LIN {X 0,Y 305.806,Z 453.018,A -85,B 0,C 180,E1 -16012.074,E2 -16012.074} C_VEL
LIN {X 0,Y 305.684,Z 453.026,A -85,B 0,C 180,E1 -16014.724,E2 -16014.724} C_VEL
LIN {X 0,Y 305.951,Z 452.995,A -85,B 0,C 180,E1 -16018.684,E2 -16018.684} C_VEL
LIN {X 0,Y 305.951,Z 452.99,A -85,B 0,C 180,E1 -16021.317,E2 -16021.317} C_VEL
LIN {X 0,Y 305.684,Z 453.027,A -85,B 0,C 180,E1 -16025.277,E2 -16025.277} C_VEL
LIN {X 0,Y 305.806,Z 453.011,A -85,B 0,C 180,E1 -16027.926,E2 -16027.926} C_VEL
LIN {X 0,Y 305.597,Z 453.04,A -85,B 0,C 180,E1 -16031.946,E2 -16031.946} C_VEL
LIN {X 0,Y 305.632,Z 453.04,A -85,B 0,C 180,E1 -16035.036,E2 -16035.036} C_VEL
LIN {X 0,Y 305.572,Z 453.044,A -85,B 0,C 180,E1 -16039.446,E2 -16039.446} C_VEL
LIN {X 0,Y 305.485,Z 453.061,A -85,B 0,C 180,E1 -16043.042,E2 -16043.042} C_VEL
LIN {X 0,Y 305.527,Z 453.043,A -85,B 0,C 180,E1 -16046.74,E2 -16046.74} C_VEL
LIN {X 0,Y 305.538,Z 453.238,A -85,B 0,C 180,E1 -16047.227,E2 -16047.227} C_VEL
LIN {X 0,Y 305.899,Z 454.626,A -85,B 0,C 180,E1 -16047.726,E2 -16047.726} C_VEL
LIN {X 0,Y 308.583,Z 458.796,A -85,B 0,C 180,E1 -16048.341,E2 -16048.341} C_VEL
LIN {X 0,Y 315.737,Z 470.32,A -85,B 0,C 180,E1 -16049.906,E2 -16049.906} C_VEL
LIN {X 0,Y 324.283,Z 485.614,A -85,B 0,C 180,E1 -16051.666,E2 -16051.666} C_VEL
LIN {X 0,Y 332.768,Z 503.328,A -85,B 0,C 180,E1 -16053.337,E2 -16053.337} C_VEL
LIN {X 0,Y 333.643,Z 505.601,A -85,B 0,C 180,E1 -16053.514,E2 -16053.514} C_VEL
LIN {X 0,Y 329.127,Z 618.858,A -85,B 0,C 180,E1 -16056.067,E2 -16056.067} C_VEL
LIN {X 0,Y 327.823,Z 634.58,A -85,B 0,C 180,E1 -16056.652,E2 -16056.652} C_VEL
LIN {X 0,Y 326.147,Z 650.125,A -85,B 0,C 180,E1 -16057.511,E2 -16057.511} C_VEL
LIN {X 0,Y 324.166,Z 664.525,A -85,B 0,C 180,E1 -16058.572,E2 -16058.572} C_VEL
LIN {X 0,Y 321.994,Z 677.479,A -85,B 0,C 180,E1 -16059.769,E2 -16059.769} C_VEL
LIN {X 0,Y 319.469,Z 690.779,A -85,B 0,C 180,E1 -16061.298,E2 -16061.298} C_VEL
LIN {X 0,Y 316.932,Z 702.653,A -85,B 0,C 180,E1 -16062.966,E2 -16062.966} C_VEL
LIN {X 0,Y 314.485,Z 713.443,A -85,B 0,C 180,E1 -16064.804,E2 -16064.804} C_VEL
LIN {X 0,Y 311.875,Z 724.247,A -85,B 0,C 180,E1 -16067.027,E2 -16067.027} C_VEL
LIN {X 0,Y 309.653,Z 733.163,A -85,B 0,C 180,E1 -16069.27,E2 -16069.27} C_VEL
LIN {X 0,Y 307.598,Z 741.721,A -85,B 0,C 180,E1 -16071.912,E2 -16071.912} C_VEL
LIN {X 0,Y 306.244,Z 747.624,A -85,B 0,C 180,E1 -16074.184,E2 -16074.184} C_VEL
LIN {X 0,Y 305.187,Z 752.434,A -85,B 0,C 180,E1 -16076.45,E2 -16076.45} C_VEL
LIN {X 0,Y 304.545,Z 756.122,A -85,B 0,C 180,E1 -16078.634,E2 -16078.634} C_VEL
LIN {X 0,Y 303.801,Z 759.699,A -85,B 0,C 180,E1 -16081.532,E2 -16081.532} C_VEL
LIN {X 0,Y 303.421,Z 761.961,A -85,B 0,C 180,E1 -16084.602,E2 -16084.602} C_VEL
LIN {X 0,Y 303.279,Z 762.664,A -85,B 0,C 180,E1 -16087.963,E2 -16087.963} C_VEL
LIN {X 0,Y 303.416,Z 761.698,A -85,B 0,C 180,E1 -16091.079,E2 -16091.079} C_VEL
LIN {X 0,Y 303.711,Z 759.497,A -85,B 0,C 180,E1 -16093.879,E2 -16093.879} C_VEL
LIN {X 0,Y 304.241,Z 756.014,A -85,B 0,C 180,E1 -16096.645,E2 -16096.645} C_VEL
LIN {X 0,Y 304.998,Z 751.21,A -85,B 0,C 180,E1 -16099.378,E2 -16099.378} C_VEL
LIN {X 0,Y 306.144,Z 744.971,A -85,B 0,C 180,E1 -16102.084,E2 -16102.084} C_VEL
LIN {X 0,Y 307.774,Z 737.108,A -85,B 0,C 180,E1 -16104.76,E2 -16104.76} C_VEL
LIN {X 0,Y 309.611,Z 728.336,A -85,B 0,C 180,E1 -16107.173,E2 -16107.173} C_VEL
LIN {X 0,Y 311.717,Z 718.677,A -85,B 0,C 180,E1 -16109.355,E2 -16109.355} C_VEL
LIN {X 0,Y 313.828,Z 708.408,A -85,B 0,C 180,E1 -16111.284,E2 -16111.284} C_VEL
LIN {X 0,Y 316.165,Z 696.881,A -85,B 0,C 180,E1 -16113.075,E2 -16113.075} C_VEL
LIN {X 0,Y 318.618,Z 683.799,A -85,B 0,C 180,E1 -16114.745,E2 -16114.745} C_VEL
LIN {X 0,Y 320.826,Z 670.4,A -85,B 0,C 180,E1 -16116.131,E2 -16116.131} C_VEL
LIN {X 0,Y 322.851,Z 655.629,A -85,B 0,C 180,E1 -16117.348,E2 -16117.348} C_VEL
LIN {X 0,Y 324.432,Z 641.335,A -85,B 0,C 180,E1 -16118.252,E2 -16118.252} C_VEL
LIN {X 0,Y 325.776,Z 625.914,A -85,B 0,C 180,E1 -16118.96,E2 -16118.96} C_VEL
LIN {X 0,Y 326.618,Z 609.669,A -85,B 0,C 180,E1 -16119.444,E2 -16119.444} C_VEL
LIN {X 0,Y 330.36,Z 503.226,A -85,B 0,C 180,E1 -16121.792,E2 -16121.792} C_VEL
LIN {X 0,Y 322.753,Z 486.044,A -85,B 0,C 180,E1 -16123.098,E2 -16123.098} C_VEL
LIN {X 0,Y 312.977,Z 466.729,A -85,B 0,C 180,E1 -16124.819,E2 -16124.819} C_VEL
LIN {X 0,Y 308.703,Z 459.164,A -85,B 0,C 180,E1 -16125.584,E2 -16125.584} C_VEL
LIN {X 0,Y 307.211,Z 456.721,A -85,B 0,C 180,E1 -16125.853,E2 -16125.853} C_VEL
LIN {X 0,Y 305.8,Z 454.164,A -85,B 0,C 180,E1 -16126.117,E2 -16126.117} C_VEL
LIN {X 0,Y 305.59,Z 453.042,A -85,B 0,C 180,E1 -16126.235,E2 -16126.235} C_VEL
LIN {X 0,Y 305.585,Z 453.048,A -85,B 0,C 180,E1 -16129.448,E2 -16129.448} C_VEL
LIN {X 0,Y 305.495,Z 453.058,A -85,B 0,C 180,E1 -16133.042,E2 -16133.042} C_VEL
LIN {X 0,Y 305.518,Z 453.047,A -85,B 0,C 180,E1 -16135.169,E2 -16135.169} C_VEL
LIN {X 0,Y 304.872,Z 453.135,A -85,B 0,C 180,E1 -16136.269,E2 -16136.269} C_VEL
LIN {X 0,Y 301.967,Z 453.492,A -85,B 0,C 180,E1 -16138.058,E2 -16138.058} C_VEL
LIN {X 0,Y 299.498,Z 453.8,A -85,B 0,C 180,E1 -16139.51,E2 -16139.51} C_VEL
LIN {X 0,Y 298.461,Z 453.933,A -85,B 0,C 180,E1 -16140.636,E2 -16140.636} C_VEL
LIN {X 0,Y 298.391,Z 453.937,A -85,B 0,C 180,E1 -16141.017,E2 -16141.017} C_VEL
LIN {X 0,Y 298.431,Z 453.936,A -85,B 0,C 180,E1 -16144.487,E2 -16144.487} C_VEL
LIN {X 0,Y 298.418,Z 453.921,A -85,B 0,C 180,E1 -16147.758,E2 -16147.758} C_VEL
LIN {X 0,Y 298.416,Z 453.939,A -85,B 0,C 180,E1 -16151.257,E2 -16151.257} C_VEL
LIN {X 0,Y 298.357,Z 453.943,A -85,B 0,C 180,E1 -16155.035,E2 -16155.035} C_VEL
LIN {X 0,Y 298.435,Z 453.934,A -85,B 0,C 180,E1 -16156.926,E2 -16156.926} C_VEL
LIN {X 0,Y 298.428,Z 453.936,A -85,B 0,C 180,E1 -16161.001,E2 -16161.001} C_VEL
LIN {X 0,Y 298.434,Z 453.921,A -85,B 0,C 180,E1 -16163.932,E2 -16163.932} C_VEL
LIN {X 0,Y 298.396,Z 453.937,A -85,B 0,C 180,E1 -16167.983,E2 -16167.983} C_VEL
LIN {X 0,Y 298.461,Z 453.926,A -85,B 0,C 180,E1 -16171.904,E2 -16171.904} C_VEL
LIN {X 0,Y 298.486,Z 453.925,A -85,B 0,C 180,E1 -16174.924,E2 -16174.924} C_VEL
LIN {X 0,Y 298.443,Z 453.932,A -85,B 0,C 180,E1 -16179.314,E2 -16179.314} C_VEL
LIN {X 0,Y 298.539,Z 453.91,A -85,B 0,C 180,E1 -16182.179,E2 -16182.179} C_VEL
LIN {X 0,Y 298.595,Z 453.905,A -85,B 0,C 180,E1 -16184.994,E2 -16184.994} C_VEL
LIN {X 0,Y 298.595,Z 453.902,A -85,B 0,C 180,E1 -16189.146,E2 -16189.146} C_VEL
LIN {X 0,Y 298.759,Z 453.885,A -85,B 0,C 180,E1 -16191.886,E2 -16191.886} C_VEL
LIN {X 0,Y 298.661,Z 453.904,A -85,B 0,C 180,E1 -16194.599,E2 -16194.599} C_VEL
LIN {X 0,Y 298.924,Z 453.867,A -85,B 0,C 180,E1 -16198.652,E2 -16198.652} C_VEL
LIN {X 0,Y 298.924,Z 453.875,A -85,B 0,C 180,E1 -16201.347,E2 -16201.347} C_VEL
LIN {X 0,Y 298.798,Z 453.883,A -85,B 0,C 180,E1 -16206.754,E2 -16206.754} C_VEL
LIN {X 0,Y 298.681,Z 453.902,A -85,B 0,C 180,E1 -16209.48,E2 -16209.48} C_VEL
LIN {X 0,Y 298.552,Z 453.909,A -85,B 0,C 180,E1 -16213.615,E2 -16213.615} C_VEL
LIN {X 0,Y 298.549,Z 453.918,A -85,B 0,C 180,E1 -16216.408,E2 -16216.408} C_VEL
LIN {X 0,Y 298.512,Z 453.911,A -85,B 0,C 180,E1 -16219.654,E2 -16219.654} C_VEL
LIN {X 0,Y 298.458,Z 453.931,A -85,B 0,C 180,E1 -16223.597,E2 -16223.597} C_VEL
LIN {X 0,Y 298.49,Z 453.928,A -85,B 0,C 180,E1 -16226.574,E2 -16226.574} C_VEL
LIN {X 0,Y 298.421,Z 453.938,A -85,B 0,C 180,E1 -16229.641,E2 -16229.641} C_VEL
LIN {X 0,Y 298.396,Z 453.939,A -85,B 0,C 180,E1 -16232.8,E2 -16232.8} C_VEL
LIN {X 0,Y 298.465,Z 453.931,A -85,B 0,C 180,E1 -16236.812,E2 -16236.812} C_VEL
LIN {X 0,Y 298.413,Z 453.938,A -85,B 0,C 180,E1 -16241.093,E2 -16241.093} C_VEL
LIN {X 0,Y 298.417,Z 453.939,A -85,B 0,C 180,E1 -16245.047,E2 -16245.047} C_VEL
LIN {X 0,Y 298.479,Z 454.134,A -85,B 0,C 180,E1 -16247.17,E2 -16247.17} C_VEL
LIN {X 0,Y 301.356,Z 464.027,A -85,B 0,C 180,E1 -16250.318,E2 -16250.318} C_VEL
LIN {X 0,Y 302.376,Z 467.643,A -85,B 0,C 180,E1 -16251.412,E2 -16251.412} C_VEL
LIN {X 0,Y 311.581,Z 486.103,A -85,B 0,C 180,E1 -16253.155,E2 -16253.155} C_VEL
LIN {X 0,Y 320.741,Z 506.44,A -85,B 0,C 180,E1 -16254.821,E2 -16254.821} C_VEL
LIN {X 0,Y 321.941,Z 509.914,A -85,B 0,C 180,E1 -16255.052,E2 -16255.052} C_VEL
LIN {X 0,Y 323.888,Z 521.419,A -85,B 0,C 180,E1 -16255.577,E2 -16255.577} C_VEL
LIN {X 0,Y 319.755,Z 634.882,A -85,B 0,C 180,E1 -16258.163,E2 -16258.163} C_VEL
LIN {X 0,Y 318.413,Z 650.708,A -85,B 0,C 180,E1 -16258.755,E2 -16258.755} C_VEL
LIN {X 0,Y 316.681,Z 665.871,A -85,B 0,C 180,E1 -16259.584,E2 -16259.584} C_VEL
LIN {X 0,Y 314.806,Z 679.599,A -85,B 0,C 180,E1 -16260.584,E2 -16260.584} C_VEL
LIN {X 0,Y 312.607,Z 693.075,A -85,B 0,C 180,E1 -16261.828,E2 -16261.828} C_VEL
LIN {X 0,Y 310.241,Z 705.501,A -85,B 0,C 180,E1 -16263.241,E2 -16263.241} C_VEL
LIN {X 0,Y 307.679,Z 718.163,A -85,B 0,C 180,E1 -16265.002,E2 -16265.002} C_VEL
LIN {X 0,Y 305.207,Z 729.668,A -85,B 0,C 180,E1 -16266.954,E2 -16266.954} C_VEL
LIN {X 0,Y 303.224,Z 739.352,A -85,B 0,C 180,E1 -16268.945,E2 -16268.945} C_VEL
LIN {X 0,Y 301.062,Z 748.848,A -85,B 0,C 180,E1 -16271.277,E2 -16271.277} C_VEL
LIN {X 0,Y 299.473,Z 756.751,A -85,B 0,C 180,E1 -16273.643,E2 -16273.643} C_VEL
LIN {X 0,Y 298.063,Z 764.116,A -85,B 0,C 180,E1 -16276.361,E2 -16276.361} C_VEL
LIN {X 0,Y 297.147,Z 769.933,A -85,B 0,C 180,E1 -16279.093,E2 -16279.093} C_VEL
LIN {X 0,Y 296.711,Z 774.37,A -85,B 0,C 180,E1 -16281.829,E2 -16281.829} C_VEL
LIN {X 0,Y 296.511,Z 777.526,A -85,B 0,C 180,E1 -16284.559,E2 -16284.559} C_VEL
LIN {X 0,Y 296.515,Z 779.449,A -85,B 0,C 180,E1 -16287.282,E2 -16287.282} C_VEL
LIN {X 0,Y 296.518,Z 780.155,A -85,B 0,C 180,E1 -16289.999,E2 -16289.999} C_VEL
LIN {X 0,Y 296.517,Z 779.71,A -85,B 0,C 180,E1 -16292.716,E2 -16292.716} C_VEL
LIN {X 0,Y 296.51,Z 778.111,A -85,B 0,C 180,E1 -16295.44,E2 -16295.44} C_VEL
LIN {X 0,Y 296.706,Z 775.339,A -85,B 0,C 180,E1 -16298.17,E2 -16298.17} C_VEL
LIN {X 0,Y 297.183,Z 771.322,A -85,B 0,C 180,E1 -16300.905,E2 -16300.905} C_VEL
LIN {X 0,Y 298.133,Z 765.949,A -85,B 0,C 180,E1 -16303.634,E2 -16303.634} C_VEL
LIN {X 0,Y 299.517,Z 759.127,A -85,B 0,C 180,E1 -16306.353,E2 -16306.353} C_VEL
LIN {X 0,Y 301.511,Z 750.68,A -85,B 0,C 180,E1 -16309.045,E2 -16309.045} C_VEL
LIN {X 0,Y 303.455,Z 743.047,A -85,B 0,C 180,E1 -16311.036,E2 -16311.036} C_VEL
LIN {X 0,Y 305.947,Z 732.701,A -85,B 0,C 180,E1 -16313.307,E2 -16313.307} C_VEL
LIN {X 0,Y 308.532,Z 721.78,A -85,B 0,C 180,E1 -16315.283,E2 -16315.283} C_VEL
LIN {X 0,Y 311.268,Z 710.08,A -85,B 0,C 180,E1 -16317.025,E2 -16317.025} C_VEL
LIN {X 0,Y 314,Z 697.34,A -85,B 0,C 180,E1 -16318.581,E2 -16318.581} C_VEL
LIN {X 0,Y 316.67,Z 683.092,A -85,B 0,C 180,E1 -16319.984,E2 -16319.984} C_VEL
LIN {X 0,Y 318.926,Z 668.805,A -85,B 0,C 180,E1 -16321.095,E2 -16321.095} C_VEL
LIN {X 0,Y 320.944,Z 653.611,A -85,B 0,C 180,E1 -16321.981,E2 -16321.981} C_VEL
LIN {X 0,Y 322.504,Z 638.634,A -85,B 0,C 180,E1 -16322.592,E2 -16322.592} C_VEL
LIN {X 0,Y 323.448,Z 620.384,A -85,B 0,C 180,E1 -16323.087,E2 -16323.087} C_VEL
LIN {X 0,Y 326.87,Z 535.782,A -85,B 0,C 180,E1 -16324.996,E2 -16324.996} C_VEL
LIN {X 0,Y 327.351,Z 521.586,A -85,B 0,C 180,E1 -16325.33,E2 -16325.33} C_VEL
LIN {X 0,Y 325.679,Z 511.869,A -85,B 0,C 180,E1 -16325.833,E2 -16325.833} C_VEL
LIN {X 0,Y 319.096,Z 497.086,A -85,B 0,C 180,E1 -16327.216,E2 -16327.216} C_VEL
LIN {X 0,Y 312.441,Z 483.929,A -85,B 0,C 180,E1 -16328.658,E2 -16328.658} C_VEL
LIN {X 0,Y 306.561,Z 473.529,A -85,B 0,C 180,E1 -16329.986,E2 -16329.986} C_VEL
LIN {X 0,Y 302.358,Z 466.202,A -85,B 0,C 180,E1 -16331.005,E2 -16331.005} C_VEL
LIN {X 0,Y 299.851,Z 458.407,A -85,B 0,C 180,E1 -16333.886,E2 -16333.886} C_VEL
LIN {X 0,Y 298.414,Z 453.93,A -85,B 0,C 180,E1 -16335.699,E2 -16335.699} C_VEL
LIN {X 0,Y 298.407,Z 453.942,A -85,B 0,C 180,E1 -16338.906,E2 -16338.906} C_VEL
LIN {X 0,Y 298.44,Z 453.936,A -85,B 0,C 180,E1 -16343.192,E2 -16343.192} C_VEL
LIN {X 0,Y 298.389,Z 453.936,A -85,B 0,C 180,E1 -16347.199,E2 -16347.199} C_VEL
LIN {X 0,Y 298.421,Z 453.934,A -85,B 0,C 180,E1 -16350.616,E2 -16350.616} C_VEL
LIN {X 0,Y 298.472,Z 453.925,A -85,B 0,C 180,E1 -16353.476,E2 -16353.476} C_VEL
LIN {X 0,Y 298.428,Z 453.931,A -85,B 0,C 180,E1 -16356.697,E2 -16356.697} C_VEL
LIN {X 0,Y 298.533,Z 453.922,A -85,B 0,C 180,E1 -16360.757,E2 -16360.757} C_VEL
LIN {X 0,Y 298.587,Z 453.917,A -85,B 0,C 180,E1 -16364.995,E2 -16364.995} C_VEL
LIN {X 0,Y 298.589,Z 453.915,A -85,B 0,C 180,E1 -16369.147,E2 -16369.147} C_VEL
LIN {X 0,Y 298.752,Z 453.895,A -85,B 0,C 180,E1 -16371.886,E2 -16371.886} C_VEL
LIN {X 0,Y 298.655,Z 453.901,A -85,B 0,C 180,E1 -16374.599,E2 -16374.599} C_VEL
LIN {X 0,Y 298.917,Z 453.871,A -85,B 0,C 180,E1 -16378.653,E2 -16378.653} C_VEL
LIN {X 0,Y 298.917,Z 453.866,A -85,B 0,C 180,E1 -16381.348,E2 -16381.348} C_VEL
LIN {X 0,Y 298.791,Z 453.891,A -85,B 0,C 180,E1 -16386.754,E2 -16386.754} C_VEL
LIN {X 0,Y 298.674,Z 453.906,A -85,B 0,C 180,E1 -16389.481,E2 -16389.481} C_VEL
LIN {X 0,Y 298.546,Z 453.918,A -85,B 0,C 180,E1 -16393.616,E2 -16393.616} C_VEL
LIN {X 0,Y 298.543,Z 453.919,A -85,B 0,C 180,E1 -16396.409,E2 -16396.409} C_VEL
LIN {X 0,Y 298.507,Z 453.925,A -85,B 0,C 180,E1 -16399.656,E2 -16399.656} C_VEL
LIN {X 0,Y 298.452,Z 453.935,A -85,B 0,C 180,E1 -16403.599,E2 -16403.599} C_VEL
LIN {X 0,Y 298.529,Z 454.023,A -85,B 0,C 180,E1 -16406.054,E2 -16406.054} C_VEL
LIN {X 0,Y 298.682,Z 454.861,A -85,B 0,C 180,E1 -16406.373,E2 -16406.373} C_VEL
LIN {X 0,Y 299.971,Z 457.462,A -85,B 0,C 180,E1 -16406.716,E2 -16406.716} C_VEL
LIN {X 0,Y 302.219,Z 460.449,A -85,B 0,C 180,E1 -16407.247,E2 -16407.247} C_VEL
LIN {X 0,Y 306.435,Z 466.935,A -85,B 0,C 180,E1 -16408.232,E2 -16408.232} C_VEL
LIN {X 0,Y 312.861,Z 477.582,A -85,B 0,C 180,E1 -16409.668,E2 -16409.668} C_VEL
LIN {X 0,Y 320.325,Z 491.438,A -85,B 0,C 180,E1 -16411.256,E2 -16411.256} C_VEL
LIN {X 0,Y 327.895,Z 507.518,A -85,B 0,C 180,E1 -16412.803,E2 -16412.803} C_VEL
LIN {X 0,Y 323.354,Z 618.445,A -85,B 0,C 180,E1 -16415.343,E2 -16415.343} C_VEL
LIN {X 0,Y 321.976,Z 634.512,A -85,B 0,C 180,E1 -16415.938,E2 -16415.938} C_VEL
LIN {X 0,Y 320.272,Z 649.718,A -85,B 0,C 180,E1 -16416.781,E2 -16416.781} C_VEL
LIN {X 0,Y 318.205,Z 664.32,A -85,B 0,C 180,E1 -16417.866,E2 -16417.866} C_VEL
LIN {X 0,Y 315.89,Z 677.646,A -85,B 0,C 180,E1 -16419.115,E2 -16419.115} C_VEL
LIN {X 0,Y 313.378,Z 690.213,A -85,B 0,C 180,E1 -16420.57,E2 -16420.57} C_VEL
LIN {X 0,Y 310.924,Z 701.391,A -85,B 0,C 180,E1 -16422.145,E2 -16422.145} C_VEL
LIN {X 0,Y 308.197,Z 712.844,A -85,B 0,C 180,E1 -16424.086,E2 -16424.086} C_VEL
LIN {X 0,Y 305.464,Z 723.795,A -85,B 0,C 180,E1 -16426.353,E2 -16426.353} C_VEL
LIN {X 0,Y 303.098,Z 732.824,A -85,B 0,C 180,E1 -16428.638,E2 -16428.638} C_VEL
LIN {X 0,Y 301.175,Z 740.331,A -85,B 0,C 180,E1 -16430.948,E2 -16430.948} C_VEL
LIN {X 0,Y 299.565,Z 746.934,A -85,B 0,C 180,E1 -16433.431,E2 -16433.431} C_VEL
LIN {X 0,Y 298.152,Z 753.058,A -85,B 0,C 180,E1 -16436.364,E2 -16436.364} C_VEL
LIN {X 0,Y 297.445,Z 756.794,A -85,B 0,C 180,E1 -16438.682,E2 -16438.682} C_VEL
LIN {X 0,Y 296.664,Z 760.277,A -85,B 0,C 180,E1 -16441.72,E2 -16441.72} C_VEL
LIN {X 0,Y 296.319,Z 762.282,A -85,B 0,C 180,E1 -16444.729,E2 -16444.729} C_VEL
LIN {X 0,Y 296.175,Z 762.896,A -85,B 0,C 180,E1 -16447.736,E2 -16447.736} C_VEL
LIN {X 0,Y 296.282,Z 762.189,A -85,B 0,C 180,E1 -16450.605,E2 -16450.605} C_VEL
LIN {X 0,Y 296.447,Z 761.343,A -85,B 0,C 180,E1 -16452.05,E2 -16452.05} C_VEL
LIN {X 0,Y 296.787,Z 758.708,A -85,B 0,C 180,E1 -16454.902,E2 -16454.902} C_VEL
LIN {X 0,Y 297.424,Z 754.78,A -85,B 0,C 180,E1 -16457.722,E2 -16457.722} C_VEL
LIN {X 0,Y 298.358,Z 749.508,A -85,B 0,C 180,E1 -16460.51,E2 -16460.51} C_VEL
LIN {X 0,Y 299.68,Z 742.773,A -85,B 0,C 180,E1 -16463.267,E2 -16463.267} C_VEL
LIN {X 0,Y 301.251,Z 735.499,A -85,B 0,C 180,E1 -16465.652,E2 -16465.652} C_VEL
LIN {X 0,Y 303.186,Z 726.696,A -85,B 0,C 180,E1 -16468.026,E2 -16468.026} C_VEL
LIN {X 0,Y 305.581,Z 716.238,A -85,B 0,C 180,E1 -16470.33,E2 -16470.33} C_VEL
LIN {X 0,Y 307.89,Z 705.466,A -85,B 0,C 180,E1 -16472.29,E2 -16472.29} C_VEL
LIN {X 0,Y 310.355,Z 693.237,A -85,B 0,C 180,E1 -16474.126,E2 -16474.126} C_VEL
LIN {X 0,Y 312.725,Z 680.865,A -85,B 0,C 180,E1 -16475.643,E2 -16475.643} C_VEL
LIN {X 0,Y 315.041,Z 666.747,A -85,B 0,C 180,E1 -16477.048,E2 -16477.048} C_VEL
LIN {X 0,Y 317.022,Z 651.966,A -85,B 0,C 180,E1 -16478.205,E2 -16478.205} C_VEL
LIN {X 0,Y 318.651,Z 636.44,A -85,B 0,C 180,E1 -16479.122,E2 -16479.122} C_VEL
LIN {X 0,Y 319.927,Z 620.693,A -85,B 0,C 180,E1 -16479.763,E2 -16479.763} C_VEL
LIN {X 0,Y 320.847,Z 599.682,A -85,B 0,C 180,E1 -16480.292,E2 -16480.292} C_VEL
LIN {X 0,Y 324.347,Z 505.684,A -85,B 0,C 180,E1 -16482.391,E2 -16482.391} C_VEL
LIN {X 0,Y 321.037,Z 497.579,A -85,B 0,C 180,E1 -16482.986,E2 -16482.986} C_VEL
LIN {X 0,Y 312.348,Z 479.314,A -85,B 0,C 180,E1 -16484.542,E2 -16484.542} C_VEL
LIN {X 0,Y 304.417,Z 464.454,A -85,B 0,C 180,E1 -16486,E2 -16486} C_VEL
LIN {X 0,Y 300.276,Z 457.77,A -85,B 0,C 180,E1 -16486.77,E2 -16486.77} C_VEL
LIN {X 0,Y 298.762,Z 454.998,A -85,B 0,C 180,E1 -16487.069,E2 -16487.069} C_VEL
LIN {X 0,Y 298.529,Z 453.925,A -85,B 0,C 180,E1 -16487.159,E2 -16487.159} C_VEL
LIN {X 0,Y 298.46,Z 453.928,A -85,B 0,C 180,E1 -16490.684,E2 -16490.684} C_VEL
LIN {X 0,Y 298.485,Z 453.922,A -85,B 0,C 180,E1 -16495.154,E2 -16495.154} C_VEL
LIN {X 0,Y 298.467,Z 453.92,A -85,B 0,C 180,E1 -16498.096,E2 -16498.096} C_VEL
LIN {X 0,Y 298.391,Z 453.937,A -85,B 0,C 180,E1 -16501.017,E2 -16501.017} C_VEL
LIN {X 0,Y 297.745,Z 454.021,A -85,B 0,C 180,E1 -16502.145,E2 -16502.145} C_VEL
LIN {X 0,Y 294.861,Z 454.379,A -85,B 0,C 180,E1 -16503.98,E2 -16503.98} C_VEL
LIN {X 0,Y 292.437,Z 454.686,A -85,B 0,C 180,E1 -16505.47,E2 -16505.47} C_VEL
LIN {X 0,Y 291.453,Z 454.798,A -85,B 0,C 180,E1 -16506.625,E2 -16506.625} C_VEL
LIN {X 0,Y 291.405,Z 454.799,A -85,B 0,C 180,E1 -16507.016,E2 -16507.016} C_VEL
LIN {X 0,Y 291.373,Z 454.815,A -85,B 0,C 180,E1 -16510.636,E2 -16510.636} C_VEL
LIN {X 0,Y 291.293,Z 454.82,A -85,B 0,C 180,E1 -16514.402,E2 -16514.402} C_VEL
LIN {X 0,Y 291.357,Z 454.802,A -85,B 0,C 180,E1 -16518.398,E2 -16518.398} C_VEL
LIN {X 0,Y 291.378,Z 454.815,A -85,B 0,C 180,E1 -16521.162,E2 -16521.162} C_VEL
LIN {X 0,Y 291.388,Z 454.8,A -85,B 0,C 180,E1 -16524.629,E2 -16524.629} C_VEL
LIN {X 0,Y 291.373,Z 454.812,A -85,B 0,C 180,E1 -16527.95,E2 -16527.95} C_VEL
LIN {X 0,Y 291.379,Z 454.801,A -85,B 0,C 180,E1 -16531.158,E2 -16531.158} C_VEL
LIN {X 0,Y 291.417,Z 454.806,A -85,B 0,C 180,E1 -16534.272,E2 -16534.272} C_VEL
LIN {X 0,Y 291.376,Z 454.795,A -85,B 0,C 180,E1 -16537.299,E2 -16537.299} C_VEL
LIN {X 0,Y 291.46,Z 454.803,A -85,B 0,C 180,E1 -16540.27,E2 -16540.27} C_VEL
LIN {X 0,Y 291.557,Z 454.78,A -85,B 0,C 180,E1 -16544.623,E2 -16544.623} C_VEL
LIN {X 0,Y 291.538,Z 454.785,A -85,B 0,C 180,E1 -16548.88,E2 -16548.88} C_VEL
LIN {X 0,Y 291.71,Z 454.76,A -85,B 0,C 180,E1 -16551.688,E2 -16551.688} C_VEL
LIN {X 0,Y 291.632,Z 454.78,A -85,B 0,C 180,E1 -16554.468,E2 -16554.468} C_VEL
LIN {X 0,Y 291.89,Z 454.743,A -85,B 0,C 180,E1 -16558.62,E2 -16558.62} C_VEL
LIN {X 0,Y 291.891,Z 454.751,A -85,B 0,C 180,E1 -16561.379,E2 -16561.379} C_VEL
LIN {X 0,Y 291.747,Z 454.762,A -85,B 0,C 180,E1 -16566.918,E2 -16566.918} C_VEL
LIN {X 0,Y 291.63,Z 454.777,A -85,B 0,C 180,E1 -16569.712,E2 -16569.712} C_VEL
LIN {X 0,Y 291.522,Z 454.788,A -85,B 0,C 180,E1 -16573.95,E2 -16573.95} C_VEL
LIN {X 0,Y 291.488,Z 454.797,A -85,B 0,C 180,E1 -16576.817,E2 -16576.817} C_VEL
LIN {X 0,Y 291.451,Z 454.793,A -85,B 0,C 180,E1 -16579.874,E2 -16579.874} C_VEL
LIN {X 0,Y 291.401,Z 454.812,A -85,B 0,C 180,E1 -16584.205,E2 -16584.205} C_VEL
LIN {X 0,Y 291.423,Z 454.81,A -85,B 0,C 180,E1 -16587.271,E2 -16587.271} C_VEL
LIN {X 0,Y 291.338,Z 454.817,A -85,B 0,C 180,E1 -16590.436,E2 -16590.436} C_VEL
LIN {X 0,Y 291.346,Z 454.816,A -85,B 0,C 180,E1 -16593.698,E2 -16593.698} C_VEL
LIN {X 0,Y 291.395,Z 454.814,A -85,B 0,C 180,E1 -16597.258,E2 -16597.258} C_VEL
LIN {X 0,Y 291.351,Z 454.816,A -85,B 0,C 180,E1 -16600.639,E2 -16600.639} C_VEL
LIN {X 0,Y 291.343,Z 454.817,A -85,B 0,C 180,E1 -16604.391,E2 -16604.391} C_VEL
LIN {X 0,Y 291.383,Z 454.927,A -85,B 0,C 180,E1 -16606.297,E2 -16606.297} C_VEL
LIN {X 0,Y 294.535,Z 465.477,A -85,B 0,C 180,E1 -16609.779,E2 -16609.779} C_VEL
LIN {X 0,Y 295.079,Z 467.572,A -85,B 0,C 180,E1 -16610.383,E2 -16610.383} C_VEL
LIN {X 0,Y 304.122,Z 485.219,A -85,B 0,C 180,E1 -16612.168,E2 -16612.168} C_VEL
LIN {X 0,Y 312.851,Z 504.176,A -85,B 0,C 180,E1 -16613.823,E2 -16613.823} C_VEL
LIN {X 0,Y 316.178,Z 512.368,A -85,B 0,C 180,E1 -16614.451,E2 -16614.451} C_VEL
LIN {X 0,Y 317.878,Z 523.572,A -85,B 0,C 180,E1 -16614.957,E2 -16614.957} C_VEL
LIN {X 0,Y 313.614,Z 634.323,A -85,B 0,C 180,E1 -16617.511,E2 -16617.511} C_VEL
LIN {X 0,Y 312.263,Z 650.291,A -85,B 0,C 180,E1 -16618.115,E2 -16618.115} C_VEL
LIN {X 0,Y 310.558,Z 664.936,A -85,B 0,C 180,E1 -16618.918,E2 -16618.918} C_VEL
LIN {X 0,Y 308.551,Z 678.97,A -85,B 0,C 180,E1 -16619.944,E2 -16619.944} C_VEL
LIN {X 0,Y 306.309,Z 692.379,A -85,B 0,C 180,E1 -16621.195,E2 -16621.195} C_VEL
LIN {X 0,Y 303.838,Z 704.902,A -85,B 0,C 180,E1 -16622.63,E2 -16622.63} C_VEL
LIN {X 0,Y 301.181,Z 717.641,A -85,B 0,C 180,E1 -16624.424,E2 -16624.424} C_VEL
LIN {X 0,Y 298.602,Z 729.207,A -85,B 0,C 180,E1 -16626.414,E2 -16626.414} C_VEL
LIN {X 0,Y 296.542,Z 738.941,A -85,B 0,C 180,E1 -16628.447,E2 -16628.447} C_VEL
LIN {X 0,Y 294.258,Z 748.472,A -85,B 0,C 180,E1 -16630.828,E2 -16630.828} C_VEL
LIN {X 0,Y 292.568,Z 756.406,A -85,B 0,C 180,E1 -16633.246,E2 -16633.246} C_VEL
LIN {X 0,Y 291.095,Z 763.8,A -85,B 0,C 180,E1 -16636.028,E2 -16636.028} C_VEL
LIN {X 0,Y 290.12,Z 769.643,A -85,B 0,C 180,E1 -16638.825,E2 -16638.825} C_VEL
LIN {X 0,Y 289.634,Z 774.104,A -85,B 0,C 180,E1 -16641.628,E2 -16641.628} C_VEL
LIN {X 0,Y 289.434,Z 777.282,A -85,B 0,C 180,E1 -16644.426,E2 -16644.426} C_VEL
LIN {X 0,Y 289.418,Z 779.216,A -85,B 0,C 180,E1 -16647.216,E2 -16647.216} C_VEL
LIN {X 0,Y 289.435,Z 779.943,A -85,B 0,C 180,E1 -16649.999,E2 -16649.999} C_VEL
LIN {X 0,Y 289.42,Z 779.516,A -85,B 0,C 180,E1 -16652.783,E2 -16652.783} C_VEL
LIN {X 0,Y 289.433,Z 777.935,A -85,B 0,C 180,E1 -16655.573,E2 -16655.573} C_VEL
LIN {X 0,Y 289.63,Z 775.182,A -85,B 0,C 180,E1 -16658.371,E2 -16658.371} C_VEL
LIN {X 0,Y 290.155,Z 771.179,A -85,B 0,C 180,E1 -16661.172,E2 -16661.172} C_VEL
LIN {X 0,Y 291.158,Z 765.832,A -85,B 0,C 180,E1 -16663.967,E2 -16663.967} C_VEL
LIN {X 0,Y 292.642,Z 759.042,A -85,B 0,C 180,E1 -16666.749,E2 -16666.749} C_VEL
LIN {X 0,Y 294.755,Z 750.623,A -85,B 0,C 180,E1 -16669.499,E2 -16669.499} C_VEL
LIN {X 0,Y 297.155,Z 741.658,A -85,B 0,C 180,E1 -16671.869,E2 -16671.869} C_VEL
LIN {X 0,Y 299.426,Z 732.546,A -85,B 0,C 180,E1 -16673.883,E2 -16673.883} C_VEL
LIN {X 0,Y 302.105,Z 721.841,A -85,B 0,C 180,E1 -16675.86,E2 -16675.86} C_VEL
LIN {X 0,Y 304.954,Z 710.217,A -85,B 0,C 180,E1 -16677.632,E2 -16677.632} C_VEL
LIN {X 0,Y 307.789,Z 697.576,A -85,B 0,C 180,E1 -16679.213,E2 -16679.213} C_VEL
LIN {X 0,Y 310.487,Z 683.829,A -85,B 0,C 180,E1 -16680.604,E2 -16680.604} C_VEL
LIN {X 0,Y 312.898,Z 669.319,A -85,B 0,C 180,E1 -16681.763,E2 -16681.763} C_VEL
LIN {X 0,Y 314.977,Z 654.38,A -85,B 0,C 180,E1 -16682.661,E2 -16682.661} C_VEL
LIN {X 0,Y 316.558,Z 639.892,A -85,B 0,C 180,E1 -16683.283,E2 -16683.283} C_VEL
LIN {X 0,Y 317.571,Z 624.127,A -85,B 0,C 180,E1 -16683.733,E2 -16683.733} C_VEL
LIN {X 0,Y 321.771,Z 523.274,A -85,B 0,C 180,E1 -16686.053,E2 -16686.053} C_VEL
LIN {X 0,Y 320.336,Z 514.663,A -85,B 0,C 180,E1 -16686.512,E2 -16686.512} C_VEL
LIN {X 0,Y 312.71,Z 497.686,A -85,B 0,C 180,E1 -16688.185,E2 -16688.185} C_VEL
LIN {X 0,Y 306.041,Z 484.836,A -85,B 0,C 180,E1 -16689.705,E2 -16689.705} C_VEL
LIN {X 0,Y 300.537,Z 475.173,A -85,B 0,C 180,E1 -16691.019,E2 -16691.019} C_VEL
LIN {X 0,Y 297.497,Z 470.211,A -85,B 0,C 180,E1 -16691.774,E2 -16691.774} C_VEL
LIN {X 0,Y 294.992,Z 465.84,A -85,B 0,C 180,E1 -16692.455,E2 -16692.455} C_VEL
LIN {X 0,Y 292.247,Z 457.43,A -85,B 0,C 180,E1 -16695.782,E2 -16695.782} C_VEL
LIN {X 0,Y 291.393,Z 454.8,A -85,B 0,C 180,E1 -16696.951,E2 -16696.951} C_VEL
LIN {X 0,Y 291.347,Z 454.82,A -85,B 0,C 180,E1 -16701.158,E2 -16701.158} C_VEL
LIN {X 0,Y 291.355,Z 454.813,A -85,B 0,C 180,E1 -16704.626,E2 -16704.626} C_VEL
LIN {X 0,Y 291.365,Z 454.814,A -85,B 0,C 180,E1 -16707.95,E2 -16707.95} C_VEL
LIN {X 0,Y 291.371,Z 454.816,A -85,B 0,C 180,E1 -16711.158,E2 -16711.158} C_VEL
LIN {X 0,Y 291.408,Z 454.811,A -85,B 0,C 180,E1 -16714.271,E2 -16714.271} C_VEL
LIN {X 0,Y 291.375,Z 454.814,A -85,B 0,C 180,E1 -16717.299,E2 -16717.299} C_VEL
LIN {X 0,Y 291.451,Z 454.799,A -85,B 0,C 180,E1 -16720.27,E2 -16720.27} C_VEL
LIN {X 0,Y 291.549,Z 454.794,A -85,B 0,C 180,E1 -16724.624,E2 -16724.624} C_VEL
LIN {X 0,Y 291.532,Z 454.795,A -85,B 0,C 180,E1 -16728.881,E2 -16728.881} C_VEL
LIN {X 0,Y 291.702,Z 454.772,A -85,B 0,C 180,E1 -16731.689,E2 -16731.689} C_VEL
LIN {X 0,Y 291.625,Z 454.776,A -85,B 0,C 180,E1 -16734.469,E2 -16734.469} C_VEL
LIN {X 0,Y 291.883,Z 454.746,A -85,B 0,C 180,E1 -16738.621,E2 -16738.621} C_VEL
LIN {X 0,Y 291.884,Z 454.742,A -85,B 0,C 180,E1 -16741.38,E2 -16741.38} C_VEL
LIN {X 0,Y 291.74,Z 454.768,A -85,B 0,C 180,E1 -16746.918,E2 -16746.918} C_VEL
LIN {X 0,Y 291.623,Z 454.785,A -85,B 0,C 180,E1 -16749.712,E2 -16749.712} C_VEL
LIN {X 0,Y 291.516,Z 454.792,A -85,B 0,C 180,E1 -16753.951,E2 -16753.951} C_VEL
LIN {X 0,Y 291.482,Z 454.798,A -85,B 0,C 180,E1 -16756.819,E2 -16756.819} C_VEL
LIN {X 0,Y 291.445,Z 454.806,A -85,B 0,C 180,E1 -16759.876,E2 -16759.876} C_VEL
LIN {X 0,Y 291.434,Z 454.815,A -85,B 0,C 180,E1 -16764.724,E2 -16764.724} C_VEL
LIN {X 0,Y 291.48,Z 455.18,A -85,B 0,C 180,E1 -16764.911,E2 -16764.911} C_VEL
LIN {X 0,Y 292.559,Z 457.843,A -85,B 0,C 180,E1 -16765.24,E2 -16765.24} C_VEL
LIN {X 0,Y 294.776,Z 460.304,A -85,B 0,C 180,E1 -16765.789,E2 -16765.789} C_VEL
LIN {X 0,Y 296.913,Z 463.61,A -85,B 0,C 180,E1 -16766.335,E2 -16766.335} C_VEL
LIN {X 0,Y 301.285,Z 470.051,A -85,B 0,C 180,E1 -16767.402,E2 -16767.402} C_VEL
LIN {X 0,Y 308.974,Z 483.088,A -85,B 0,C 180,E1 -16769.197,E2 -16769.197} C_VEL
LIN {X 0,Y 316.136,Z 496.677,A -85,B 0,C 180,E1 -16770.779,E2 -16770.779} C_VEL
LIN {X 0,Y 322.266,Z 509.845,A -85,B 0,C 180,E1 -16772.083,E2 -16772.083} C_VEL
LIN {X 0,Y 317.557,Z 618.874,A -85,B 0,C 180,E1 -16774.615,E2 -16774.615} C_VEL
LIN {X 0,Y 316.163,Z 634.673,A -85,B 0,C 180,E1 -16775.21,E2 -16775.21} C_VEL
LIN {X 0,Y 314.353,Z 650.091,A -85,B 0,C 180,E1 -16776.076,E2 -16776.076} C_VEL
LIN {X 0,Y 312.242,Z 664.552,A -85,B 0,C 180,E1 -16777.169,E2 -16777.169} C_VEL
LIN {X 0,Y 309.727,Z 678.313,A -85,B 0,C 180,E1 -16778.481,E2 -16778.481} C_VEL
LIN {X 0,Y 307.112,Z 690.864,A -85,B 0,C 180,E1 -16779.966,E2 -16779.966} C_VEL
LIN {X 0,Y 304.17,Z 703.627,A -85,B 0,C 180,E1 -16781.831,E2 -16781.831} C_VEL
LIN {X 0,Y 301.492,Z 714.317,A -85,B 0,C 180,E1 -16783.729,E2 -16783.729} C_VEL
LIN {X 0,Y 298.659,Z 725.034,A -85,B 0,C 180,E1 -16786.039,E2 -16786.039} C_VEL
LIN {X 0,Y 296.227,Z 733.895,A -85,B 0,C 180,E1 -16788.373,E2 -16788.373} C_VEL
LIN {X 0,Y 293.928,Z 742.371,A -85,B 0,C 180,E1 -16791.124,E2 -16791.124} C_VEL
LIN {X 0,Y 292.198,Z 749.133,A -85,B 0,C 180,E1 -16793.896,E2 -16793.896} C_VEL
LIN {X 0,Y 290.827,Z 755.019,A -85,B 0,C 180,E1 -16797.065,E2 -16797.065} C_VEL
LIN {X 0,Y 290.117,Z 758.286,A -85,B 0,C 180,E1 -16799.423,E2 -16799.423} C_VEL
LIN {X 0,Y 289.456,Z 761.28,A -85,B 0,C 180,E1 -16802.529,E2 -16802.529} C_VEL
LIN {X 0,Y 289.137,Z 762.819,A -85,B 0,C 180,E1 -16805.594,E2 -16805.594} C_VEL
LIN {X 0,Y 289.084,Z 762.988,A -85,B 0,C 180,E1 -16808.614,E2 -16808.614} C_VEL
LIN {X 0,Y 289.323,Z 761.847,A -85,B 0,C 180,E1 -16811.593,E2 -16811.593} C_VEL
LIN {X 0,Y 289.611,Z 759.446,A -85,B 0,C 180,E1 -16814.519,E2 -16814.519} C_VEL
LIN {X 0,Y 290.252,Z 755.752,A -85,B 0,C 180,E1 -16817.414,E2 -16817.414} C_VEL
LIN {X 0,Y 291.159,Z 750.729,A -85,B 0,C 180,E1 -16820.273,E2 -16820.273} C_VEL
LIN {X 0,Y 292.498,Z 744.253,A -85,B 0,C 180,E1 -16823.101,E2 -16823.101} C_VEL
LIN {X 0,Y 294.063,Z 737.271,A -85,B 0,C 180,E1 -16825.546,E2 -16825.546} C_VEL
LIN {X 0,Y 296.089,Z 728.484,A -85,B 0,C 180,E1 -16828.053,E2 -16828.053} C_VEL
LIN {X 0,Y 298.383,Z 718.709,A -85,B 0,C 180,E1 -16830.338,E2 -16830.338} C_VEL
LIN {X 0,Y 300.737,Z 708.357,A -85,B 0,C 180,E1 -16832.345,E2 -16832.345} C_VEL
LIN {X 0,Y 303.41,Z 695.893,A -85,B 0,C 180,E1 -16834.327,E2 -16834.327} C_VEL
LIN {X 0,Y 305.89,Z 683.522,A -85,B 0,C 180,E1 -16835.935,E2 -16835.935} C_VEL
LIN {X 0,Y 308.278,Z 669.953,A -85,B 0,C 180,E1 -16837.368,E2 -16837.368} C_VEL
LIN {X 0,Y 310.308,Z 655.974,A -85,B 0,C 180,E1 -16838.548,E2 -16838.548} C_VEL
LIN {X 0,Y 312.017,Z 641.64,A -85,B 0,C 180,E1 -16839.481,E2 -16839.481} C_VEL
LIN {X 0,Y 313.411,Z 626.23,A -85,B 0,C 180,E1 -16840.213,E2 -16840.213} C_VEL
LIN {X 0,Y 314.343,Z 609.996,A -85,B 0,C 180,E1 -16840.707,E2 -16840.707} C_VEL
LIN {X 0,Y 318.262,Z 507.166,A -85,B 0,C 180,E1 -16843.048,E2 -16843.048} C_VEL
LIN {X 0,Y 310.362,Z 489.633,A -85,B 0,C 180,E1 -16844.499,E2 -16844.499} C_VEL
LIN {X 0,Y 300.197,Z 469.753,A -85,B 0,C 180,E1 -16846.42,E2 -16846.42} C_VEL
LIN {X 0,Y 293.962,Z 459.514,A -85,B 0,C 180,E1 -16847.629,E2 -16847.629} C_VEL
LIN {X 0,Y 291.964,Z 456.55,A -85,B 0,C 180,E1 -16848.016,E2 -16848.016} C_VEL
LIN {X 0,Y 291.5,Z 454.795,A -85,B 0,C 180,E1 -16848.176,E2 -16848.176} C_VEL
LIN {X 0,Y 291.385,Z 454.808,A -85,B 0,C 180,E1 -16851.211,E2 -16851.211} C_VEL
LIN {X 0,Y 291.404,Z 454.802,A -85,B 0,C 180,E1 -16854.205,E2 -16854.205} C_VEL
LIN {X 0,Y 291.427,Z 454.801,A -85,B 0,C 180,E1 -16857.272,E2 -16857.272} C_VEL
LIN {X 0,Y 291.327,Z 454.814,A -85,B 0,C 180,E1 -16861.018,E2 -16861.018} C_VEL
LIN {X 0,Y 291.365,Z 454.819,A -85,B 0,C 180,E1 -16865.374,E2 -16865.374} C_VEL
LIN {X 0,Y 291.405,Z 454.799,A -85,B 0,C 180,E1 -16867.016,E2 -16867.016} C_VEL
LIN {X 0,Y 291.145,Z 454.832,A -85,B 0,C 180,E1 -16867.786,E2 -16867.786} C_VEL
LIN {X 0,Y 289.819,Z 455.003,A -85,B 0,C 180,E1 -16868.923,E2 -16868.923} C_VEL
LIN {X 0,Y 285.404,Z 455.557,A -85,B 0,C 180,E1 -16871.563,E2 -16871.563} C_VEL
LIN {X 0,Y 284.325,Z 455.683,A -85,B 0,C 180,E1 -16872.744,E2 -16872.744} C_VEL
LIN {X 0,Y 284.24,Z 455.691,A -85,B 0,C 180,E1 -16873.144,E2 -16873.144} C_VEL
LIN {X 0,Y 284.275,Z 455.698,A -85,B 0,C 180,E1 -16876.192,E2 -16876.192} C_VEL
LIN {X 0,Y 284.354,Z 455.685,A -85,B 0,C 180,E1 -16880.013,E2 -16880.013} C_VEL
LIN {X 0,Y 284.354,Z 455.675,A -85,B 0,C 180,E1 -16883.617,E2 -16883.617} C_VEL
LIN {X 0,Y 284.31,Z 455.695,A -85,B 0,C 180,E1 -16887.189,E2 -16887.189} C_VEL
LIN {X 0,Y 284.357,Z 455.671,A -85,B 0,C 180,E1 -16890.375,E2 -16890.375} C_VEL
LIN {X 0,Y 284.379,Z 455.689,A -85,B 0,C 180,E1 -16893.586,E2 -16893.586} C_VEL
LIN {X 0,Y 284.335,Z 455.67,A -85,B 0,C 180,E1 -16896.704,E2 -16896.704} C_VEL
LIN {X 0,Y 284.405,Z 455.679,A -85,B 0,C 180,E1 -16901.261,E2 -16901.261} C_VEL
LIN {X 0,Y 284.494,Z 455.657,A -85,B 0,C 180,E1 -16904.459,E2 -16904.459} C_VEL
LIN {X 0,Y 284.49,Z 455.664,A -85,B 0,C 180,E1 -16908.601,E2 -16908.601} C_VEL
LIN {X 0,Y 284.66,Z 455.636,A -85,B 0,C 180,E1 -16911.481,E2 -16911.481} C_VEL
LIN {X 0,Y 284.603,Z 455.656,A -85,B 0,C 180,E1 -16914.331,E2 -16914.331} C_VEL
LIN {X 0,Y 284.856,Z 455.618,A -85,B 0,C 180,E1 -16918.586,E2 -16918.586} C_VEL
LIN {X 0,Y 284.857,Z 455.626,A -85,B 0,C 180,E1 -16921.413,E2 -16921.413} C_VEL
LIN {X 0,Y 284.699,Z 455.64,A -85,B 0,C 180,E1 -16927.09,E2 -16927.09} C_VEL
LIN {X 0,Y 284.568,Z 455.654,A -85,B 0,C 180,E1 -16929.955,E2 -16929.955} C_VEL
LIN {X 0,Y 284.482,Z 455.67,A -85,B 0,C 180,E1 -16934.302,E2 -16934.302} C_VEL
LIN {X 0,Y 284.426,Z 455.669,A -85,B 0,C 180,E1 -16937.248,E2 -16937.248} C_VEL
LIN {X 0,Y 284.381,Z 455.679,A -85,B 0,C 180,E1 -16940.242,E2 -16940.242} C_VEL
LIN {X 0,Y 284.37,Z 455.688,A -85,B 0,C 180,E1 -16943.875,E2 -16943.875} C_VEL
LIN {X 0,Y 284.398,Z 455.684,A -85,B 0,C 180,E1 -16947.173,E2 -16947.173} C_VEL
LIN {X 0,Y 284.297,Z 455.693,A -85,B 0,C 180,E1 -16951.274,E2 -16951.274} C_VEL
LIN {X 0,Y 284.362,Z 455.687,A -85,B 0,C 180,E1 -16955.353,E2 -16955.353} C_VEL
LIN {X 0,Y 284.324,Z 455.691,A -85,B 0,C 180,E1 -16958.167,E2 -16958.167} C_VEL
LIN {X 0,Y 284.297,Z 455.695,A -85,B 0,C 180,E1 -16962.13,E2 -16962.13} C_VEL
LIN {X 0,Y 284.337,Z 455.81,A -85,B 0,C 180,E1 -16965.411,E2 -16965.411} C_VEL
LIN {X 0,Y 287.181,Z 465.205,A -85,B 0,C 180,E1 -16968.642,E2 -16968.642} C_VEL
LIN {X 0,Y 287.789,Z 467.322,A -85,B 0,C 180,E1 -16969.288,E2 -16969.288} C_VEL
LIN {X 0,Y 297.535,Z 486.06,A -85,B 0,C 180,E1 -16971.298,E2 -16971.298} C_VEL
LIN {X 0,Y 306.408,Z 505.191,A -85,B 0,C 180,E1 -16973.046,E2 -16973.046} C_VEL
LIN {X 0,Y 310.488,Z 514.985,A -85,B 0,C 180,E1 -16973.837,E2 -16973.837} C_VEL
LIN {X 0,Y 311.895,Z 524.386,A -85,B 0,C 180,E1 -16974.273,E2 -16974.273} C_VEL
LIN {X 0,Y 307.508,Z 633.71,A -85,B 0,C 180,E1 -16976.832,E2 -16976.832} C_VEL
LIN {X 0,Y 306.155,Z 649.856,A -85,B 0,C 180,E1 -16977.45,E2 -16977.45} C_VEL
LIN {X 0,Y 304.285,Z 665.132,A -85,B 0,C 180,E1 -16978.301,E2 -16978.301} C_VEL
LIN {X 0,Y 302.135,Z 679.63,A -85,B 0,C 180,E1 -16979.39,E2 -16979.39} C_VEL
LIN {X 0,Y 299.759,Z 693.228,A -85,B 0,C 180,E1 -16980.697,E2 -16980.697} C_VEL
LIN {X 0,Y 296.98,Z 706.837,A -85,B 0,C 180,E1 -16982.327,E2 -16982.327} C_VEL
LIN {X 0,Y 294.255,Z 719.212,A -85,B 0,C 180,E1 -16984.158,E2 -16984.158} C_VEL
LIN {X 0,Y 291.628,Z 730.453,A -85,B 0,C 180,E1 -16986.182,E2 -16986.182} C_VEL
LIN {X 0,Y 289.133,Z 741.448,A -85,B 0,C 180,E1 -16988.616,E2 -16988.616} C_VEL
LIN {X 0,Y 286.937,Z 750.545,A -85,B 0,C 180,E1 -16991.062,E2 -16991.062} C_VEL
LIN {X 0,Y 285.216,Z 758.297,A -85,B 0,C 180,E1 -16993.611,E2 -16993.611} C_VEL
LIN {X 0,Y 283.86,Z 765.114,A -85,B 0,C 180,E1 -16996.396,E2 -16996.396} C_VEL
LIN {X 0,Y 282.927,Z 770.611,A -85,B 0,C 180,E1 -16999.262,E2 -16999.262} C_VEL
LIN {X 0,Y 282.579,Z 773.837,A -85,B 0,C 180,E1 -17001.417,E2 -17001.417} C_VEL
LIN {X 0,Y 282.34,Z 777.038,A -85,B 0,C 180,E1 -17004.285,E2 -17004.285} C_VEL
LIN {X 0,Y 282.324,Z 778.983,A -85,B 0,C 180,E1 -17007.145,E2 -17007.145} C_VEL
LIN {X 0,Y 282.355,Z 779.73,A -85,B 0,C 180,E1 -17009.999,E2 -17009.999} C_VEL
LIN {X 0,Y 282.326,Z 779.322,A -85,B 0,C 180,E1 -17012.853,E2 -17012.853} C_VEL
LIN {X 0,Y 282.339,Z 777.763,A -85,B 0,C 180,E1 -17015.713,E2 -17015.713} C_VEL
LIN {X 0,Y 282.571,Z 775.035,A -85,B 0,C 180,E1 -17018.581,E2 -17018.581} C_VEL
LIN {X 0,Y 283.133,Z 771.044,A -85,B 0,C 180,E1 -17021.453,E2 -17021.453} C_VEL
LIN {X 0,Y 284.202,Z 765.721,A -85,B 0,C 180,E1 -17024.316,E2 -17024.316} C_VEL
LIN {X 0,Y 285.778,Z 758.956,A -85,B 0,C 180,E1 -17027.163,E2 -17027.163} C_VEL
LIN {X 0,Y 288.005,Z 750.565,A -85,B 0,C 180,E1 -17029.975,E2 -17029.975} C_VEL
LIN {X 0,Y 290.537,Z 741.646,A -85,B 0,C 180,E1 -17032.394,E2 -17032.394} C_VEL
LIN {X 0,Y 293.323,Z 730.958,A -85,B 0,C 180,E1 -17034.789,E2 -17034.789} C_VEL
LIN {X 0,Y 296.271,Z 719.993,A -85,B 0,C 180,E1 -17036.788,E2 -17036.788} C_VEL
LIN {X 0,Y 299.248,Z 708.041,A -85,B 0,C 180,E1 -17038.587,E2 -17038.587} C_VEL
LIN {X 0,Y 302.226,Z 694.981,A -85,B 0,C 180,E1 -17040.189,E2 -17040.189} C_VEL
LIN {X 0,Y 304.913,Z 681.348,A -85,B 0,C 180,E1 -17041.539,E2 -17041.539} C_VEL
LIN {X 0,Y 307.406,Z 666.484,A -85,B 0,C 180,E1 -17042.691,E2 -17042.691} C_VEL
LIN {X 0,Y 309.484,Z 652.144,A -85,B 0,C 180,E1 -17043.51,E2 -17043.51} C_VEL
LIN {X 0,Y 311.047,Z 636.744,A -85,B 0,C 180,E1 -17044.147,E2 -17044.147} C_VEL
LIN {X 0,Y 312.166,Z 616.112,A -85,B 0,C 180,E1 -17044.691,E2 -17044.691} C_VEL
LIN {X 0,Y 315.639,Z 537.854,A -85,B 0,C 180,E1 -17046.512,E2 -17046.512} C_VEL
LIN {X 0,Y 316.169,Z 524.009,A -85,B 0,C 180,E1 -17046.848,E2 -17046.848} C_VEL
LIN {X 0,Y 315.07,Z 517.641,A -85,B 0,C 180,E1 -17047.205,E2 -17047.205} C_VEL
LIN {X 0,Y 307.536,Z 500.775,A -85,B 0,C 180,E1 -17048.933,E2 -17048.933} C_VEL
LIN {X 0,Y 301.692,Z 489.402,A -85,B 0,C 180,E1 -17050.324,E2 -17050.324} C_VEL
LIN {X 0,Y 296.18,Z 479.6,A -85,B 0,C 180,E1 -17051.699,E2 -17051.699} C_VEL
LIN {X 0,Y 290.342,Z 470.068,A -85,B 0,C 180,E1 -17053.232,E2 -17053.232} C_VEL
LIN {X 0,Y 287.615,Z 465.575,A -85,B 0,C 180,E1 -17054.007,E2 -17054.007} C_VEL
LIN {X 0,Y 285.047,Z 457.988,A -85,B 0,C 180,E1 -17057.238,E2 -17057.238} C_VEL
LIN {X 0,Y 284.312,Z 455.697,A -85,B 0,C 180,E1 -17058.369,E2 -17058.369} C_VEL
LIN {X 0,Y 284.317,Z 455.691,A -85,B 0,C 180,E1 -17062.277,E2 -17062.277} C_VEL
LIN {X 0,Y 284.303,Z 455.696,A -85,B 0,C 180,E1 -17065.35,E2 -17065.35} C_VEL
LIN {X 0,Y 284.288,Z 455.698,A -85,B 0,C 180,E1 -17068.725,E2 -17068.725} C_VEL
LIN {X 0,Y 284.389,Z 455.678,A -85,B 0,C 180,E1 -17072.827,E2 -17072.827} C_VEL
LIN {X 0,Y 284.36,Z 455.683,A -85,B 0,C 180,E1 -17076.707,E2 -17076.707} C_VEL
LIN {X 0,Y 284.397,Z 455.685,A -85,B 0,C 180,E1 -17081.262,E2 -17081.262} C_VEL
LIN {X 0,Y 284.486,Z 455.671,A -85,B 0,C 180,E1 -17084.459,E2 -17084.459} C_VEL
LIN {X 0,Y 284.483,Z 455.675,A -85,B 0,C 180,E1 -17088.602,E2 -17088.602} C_VEL
LIN {X 0,Y 284.653,Z 455.649,A -85,B 0,C 180,E1 -17091.481,E2 -17091.481} C_VEL
LIN {X 0,Y 284.596,Z 455.651,A -85,B 0,C 180,E1 -17094.332,E2 -17094.332} C_VEL
LIN {X 0,Y 284.85,Z 455.622,A -85,B 0,C 180,E1 -17098.587,E2 -17098.587} C_VEL
LIN {X 0,Y 284.85,Z 455.618,A -85,B 0,C 180,E1 -17101.414,E2 -17101.414} C_VEL
LIN {X 0,Y 284.692,Z 455.646,A -85,B 0,C 180,E1 -17107.091,E2 -17107.091} C_VEL
LIN {X 0,Y 284.561,Z 455.665,A -85,B 0,C 180,E1 -17109.956,E2 -17109.956} C_VEL
LIN {X 0,Y 284.476,Z 455.669,A -85,B 0,C 180,E1 -17114.303,E2 -17114.303} C_VEL
LIN {X 0,Y 284.42,Z 455.679,A -85,B 0,C 180,E1 -17117.249,E2 -17117.249} C_VEL
LIN {X 0,Y 284.374,Z 455.69,A -85,B 0,C 180,E1 -17120.243,E2 -17120.243} C_VEL
LIN {X 0,Y 284.382,Z 455.824,A -85,B 0,C 180,E1 -17123.346,E2 -17123.346} C_VEL
LIN {X 0,Y 285.329,Z 458.467,A -85,B 0,C 180,E1 -17123.674,E2 -17123.674} C_VEL
LIN {X 0,Y 287.368,Z 460.663,A -85,B 0,C 180,E1 -17124.221,E2 -17124.221} C_VEL
LIN {X 0,Y 290.293,Z 464.852,A -85,B 0,C 180,E1 -17125.019,E2 -17125.019} C_VEL
LIN {X 0,Y 291.757,Z 466.958,A -85,B 0,C 180,E1 -17125.409,E2 -17125.409} C_VEL
LIN {X 0,Y 297.046,Z 474.579,A -85,B 0,C 180,E1 -17126.749,E2 -17126.749} C_VEL
LIN {X 0,Y 304.64,Z 487.684,A -85,B 0,C 180,E1 -17128.602,E2 -17128.602} C_VEL
LIN {X 0,Y 312.184,Z 502.283,A -85,B 0,C 180,E1 -17130.333,E2 -17130.333} C_VEL
LIN {X 0,Y 316.68,Z 512.172,A -85,B 0,C 180,E1 -17131.33,E2 -17131.33} C_VEL
LIN {X 0,Y 311.808,Z 619.414,A -85,B 0,C 180,E1 -17133.858,E2 -17133.858} C_VEL
LIN {X 0,Y 310.416,Z 634.756,A -85,B 0,C 180,E1 -17134.448,E2 -17134.448} C_VEL
LIN {X 0,Y 308.513,Z 650.325,A -85,B 0,C 180,E1 -17135.334,E2 -17135.334} C_VEL
LIN {X 0,Y 306.316,Z 664.793,A -85,B 0,C 180,E1 -17136.444,E2 -17136.444} C_VEL
LIN {X 0,Y 303.617,Z 678.986,A -85,B 0,C 180,E1 -17137.825,E2 -17137.825} C_VEL
LIN {X 0,Y 300.886,Z 691.549,A -85,B 0,C 180,E1 -17139.345,E2 -17139.345} C_VEL
LIN {X 0,Y 297.733,Z 704.511,A -85,B 0,C 180,E1 -17141.288,E2 -17141.288} C_VEL
LIN {X 0,Y 294.861,Z 715.441,A -85,B 0,C 180,E1 -17143.29,E2 -17143.29} C_VEL
LIN {X 0,Y 291.865,Z 726.222,A -85,B 0,C 180,E1 -17145.71,E2 -17145.71} C_VEL
LIN {X 0,Y 289.351,Z 734.924,A -85,B 0,C 180,E1 -17148.093,E2 -17148.093} C_VEL
LIN {X 0,Y 287.301,Z 742.153,A -85,B 0,C 180,E1 -17150.506,E2 -17150.506} C_VEL
LIN {X 0,Y 285.659,Z 748.091,A -85,B 0,C 180,E1 -17152.933,E2 -17152.933} C_VEL
LIN {X 0,Y 284.388,Z 752.941,A -85,B 0,C 180,E1 -17155.363,E2 -17155.363} C_VEL
LIN {X 0,Y 283.635,Z 756.201,A -85,B 0,C 180,E1 -17157.402,E2 -17157.402} C_VEL
LIN {X 0,Y 282.762,Z 759.884,A -85,B 0,C 180,E1 -17160.45,E2 -17160.45} C_VEL
LIN {X 0,Y 282.212,Z 762.321,A -85,B 0,C 180,E1 -17163.705,E2 -17163.705} C_VEL
LIN {X 0,Y 281.989,Z 763.226,A -85,B 0,C 180,E1 -17166.5,E2 -17166.5} C_VEL
LIN {X 0,Y 282.014,Z 762.97,A -85,B 0,C 180,E1 -17169.582,E2 -17169.582} C_VEL
LIN {X 0,Y 282.179,Z 762.321,A -85,B 0,C 180,E1 -17171.164,E2 -17171.164} C_VEL
LIN {X 0,Y 282.457,Z 760.18,A -85,B 0,C 180,E1 -17174.117,E2 -17174.117} C_VEL
LIN {X 0,Y 283.087,Z 756.718,A -85,B 0,C 180,E1 -17177.09,E2 -17177.09} C_VEL
LIN {X 0,Y 283.962,Z 751.935,A -85,B 0,C 180,E1 -17180.024,E2 -17180.024} C_VEL
LIN {X 0,Y 285.285,Z 745.718,A -85,B 0,C 180,E1 -17182.925,E2 -17182.925} C_VEL
LIN {X 0,Y 287.123,Z 737.888,A -85,B 0,C 180,E1 -17185.79,E2 -17185.79} C_VEL
LIN {X 0,Y 289.18,Z 729.304,A -85,B 0,C 180,E1 -17188.324,E2 -17188.324} C_VEL
LIN {X 0,Y 291.582,Z 719.5,A -85,B 0,C 180,E1 -17190.691,E2 -17190.691} C_VEL
LIN {X 0,Y 294.001,Z 709.223,A -85,B 0,C 180,E1 -17192.741,E2 -17192.741} C_VEL
LIN {X 0,Y 296.682,Z 697.145,A -85,B 0,C 180,E1 -17194.733,E2 -17194.733} C_VEL
LIN {X 0,Y 299.334,Z 684.665,A -85,B 0,C 180,E1 -17196.404,E2 -17196.404} C_VEL
LIN {X 0,Y 301.762,Z 671.318,A -85,B 0,C 180,E1 -17197.865,E2 -17197.865} C_VEL
LIN {X 0,Y 303.996,Z 656.625,A -85,B 0,C 180,E1 -17199.146,E2 -17199.146} C_VEL
LIN {X 0,Y 305.778,Z 642.396,A -85,B 0,C 180,E1 -17200.094,E2 -17200.094} C_VEL
LIN {X 0,Y 307.197,Z 627.237,A -85,B 0,C 180,E1 -17200.839,E2 -17200.839} C_VEL
LIN {X 0,Y 308.096,Z 612.743,A -85,B 0,C 180,E1 -17201.311,E2 -17201.311} C_VEL
LIN {X 0,Y 312.265,Z 509.242,A -85,B 0,C 180,E1 -17203.708,E2 -17203.708} C_VEL
LIN {X 0,Y 304.415,Z 491.819,A -85,B 0,C 180,E1 -17205.196,E2 -17205.196} C_VEL
LIN {X 0,Y 295.157,Z 473.848,A -85,B 0,C 180,E1 -17207.009,E2 -17207.009} C_VEL
LIN {X 0,Y 286.345,Z 459.73,A -85,B 0,C 180,E1 -17208.771,E2 -17208.771} C_VEL
LIN {X 0,Y 284.817,Z 457.334,A -85,B 0,C 180,E1 -17209.09,E2 -17209.09} C_VEL
LIN {X 0,Y 284.423,Z 455.683,A -85,B 0,C 180,E1 -17209.23,E2 -17209.23} C_VEL
LIN {X 0,Y 284.373,Z 455.679,A -85,B 0,C 180,E1 -17213.876,E2 -17213.876} C_VEL
LIN {X 0,Y 284.401,Z 455.677,A -85,B 0,C 180,E1 -17217.174,E2 -17217.174} C_VEL
LIN {X 0,Y 284.3,Z 455.691,A -85,B 0,C 180,E1 -17221.274,E2 -17221.274} C_VEL
LIN {X 0,Y 284.345,Z 455.694,A -85,B 0,C 180,E1 -17225.348,E2 -17225.348} C_VEL
LIN {X 0,Y 284.316,Z 455.676,A -85,B 0,C 180,E1 -17228.169,E2 -17228.169} C_VEL
LIN {X 0,Y 284.292,Z 455.693,A -85,B 0,C 180,E1 -17231.872,E2 -17231.872} C_VEL
LIN {X 0,Y 284.24,Z 455.691,A -85,B 0,C 180,E1 -17233.144,E2 -17233.144} C_VEL
LIN {X 0,Y 283.572,Z 455.781,A -85,B 0,C 180,E1 -17234.328,E2 -17234.328} C_VEL
LIN {X 0,Y 280.713,Z 456.142,A -85,B 0,C 180,E1 -17236.256,E2 -17236.256} C_VEL
LIN {X 0,Y 278.312,Z 456.431,A -85,B 0,C 180,E1 -17237.823,E2 -17237.823} C_VEL
LIN {X 0,Y 277.321,Z 456.552,A -85,B 0,C 180,E1 -17239.037,E2 -17239.037} C_VEL
LIN {X 0,Y 277.261,Z 456.562,A -85,B 0,C 180,E1 -17239.448,E2 -17239.448} C_VEL
LIN {X 0,Y 277.288,Z 456.564,A -85,B 0,C 180,E1 -17242.533,E2 -17242.533} C_VEL
LIN {X 0,Y 277.257,Z 456.572,A -85,B 0,C 180,E1 -17246.105,E2 -17246.105} C_VEL
LIN {X 0,Y 277.264,Z 456.556,A -85,B 0,C 180,E1 -17249.538,E2 -17249.538} C_VEL
LIN {X 0,Y 277.36,Z 456.559,A -85,B 0,C 180,E1 -17252.864,E2 -17252.864} C_VEL
LIN {X 0,Y 277.299,Z 456.548,A -85,B 0,C 180,E1 -17256.076,E2 -17256.076} C_VEL
LIN {X 0,Y 277.347,Z 456.56,A -85,B 0,C 180,E1 -17260.766,E2 -17260.766} C_VEL
LIN {X 0,Y 277.436,Z 456.542,A -85,B 0,C 180,E1 -17265.326,E2 -17265.326} C_VEL
LIN {X 0,Y 277.508,Z 456.522,A -85,B 0,C 180,E1 -17269.788,E2 -17269.788} C_VEL
LIN {X 0,Y 277.654,Z 456.52,A -85,B 0,C 180,E1 -17272.729,E2 -17272.729} C_VEL
LIN {X 0,Y 277.822,Z 456.493,A -85,B 0,C 180,E1 -17278.55,E2 -17278.55} C_VEL
LIN {X 0,Y 277.823,Z 456.502,A -85,B 0,C 180,E1 -17281.449,E2 -17281.449} C_VEL
LIN {X 0,Y 277.654,Z 456.519,A -85,B 0,C 180,E1 -17287.271,E2 -17287.271} C_VEL
LIN {X 0,Y 277.508,Z 456.532,A -85,B 0,C 180,E1 -17290.211,E2 -17290.211} C_VEL
LIN {X 0,Y 277.435,Z 456.549,A -85,B 0,C 180,E1 -17294.674,E2 -17294.674} C_VEL
LIN {X 0,Y 277.346,Z 456.543,A -85,B 0,C 180,E1 -17299.233,E2 -17299.233} C_VEL
LIN {X 0,Y 277.33,Z 456.565,A -85,B 0,C 180,E1 -17303.92,E2 -17303.92} C_VEL
LIN {X 0,Y 277.327,Z 456.565,A -85,B 0,C 180,E1 -17307.505,E2 -17307.505} C_VEL
LIN {X 0,Y 277.273,Z 456.569,A -85,B 0,C 180,E1 -17310.481,E2 -17310.481} C_VEL
LIN {X 0,Y 277.255,Z 456.572,A -85,B 0,C 180,E1 -17313.894,E2 -17313.894} C_VEL
LIN {X 0,Y 277.282,Z 456.57,A -85,B 0,C 180,E1 -17317.467,E2 -17317.467} C_VEL
LIN {X 0,Y 277.227,Z 456.578,A -85,B 0,C 180,E1 -17321.233,E2 -17321.233} C_VEL
LIN {X 0,Y 277.283,Z 456.772,A -85,B 0,C 180,E1 -17324.501,E2 -17324.501} C_VEL
LIN {X 0,Y 280.484,Z 467.088,A -85,B 0,C 180,E1 -17328.128,E2 -17328.128} C_VEL
LIN {X 0,Y 290.693,Z 486.398,A -85,B 0,C 180,E1 -17330.331,E2 -17330.331} C_VEL
LIN {X 0,Y 299.219,Z 504.452,A -85,B 0,C 180,E1 -17332.083,E2 -17332.083} C_VEL
LIN {X 0,Y 304.838,Z 517.83,A -85,B 0,C 180,E1 -17333.211,E2 -17333.211} C_VEL
LIN {X 0,Y 305.931,Z 525.8,A -85,B 0,C 180,E1 -17333.579,E2 -17333.579} C_VEL
LIN {X 0,Y 301.394,Z 634.394,A -85,B 0,C 180,E1 -17336.17,E2 -17336.17} C_VEL
LIN {X 0,Y 299.963,Z 650.18,A -85,B 0,C 180,E1 -17336.793,E2 -17336.793} C_VEL
LIN {X 0,Y 298.067,Z 665.321,A -85,B 0,C 180,E1 -17337.66,E2 -17337.66} C_VEL
LIN {X 0,Y 295.998,Z 678.812,A -85,B 0,C 180,E1 -17338.684,E2 -17338.684} C_VEL
LIN {X 0,Y 293.536,Z 692.52,A -85,B 0,C 180,E1 -17340.013,E2 -17340.013} C_VEL
LIN {X 0,Y 290.627,Z 706.234,A -85,B 0,C 180,E1 -17341.668,E2 -17341.668} C_VEL
LIN {X 0,Y 287.8,Z 718.676,A -85,B 0,C 180,E1 -17343.534,E2 -17343.534} C_VEL
LIN {X 0,Y 285.119,Z 729.784,A -85,B 0,C 180,E1 -17345.564,E2 -17345.564} C_VEL
LIN {X 0,Y 282.861,Z 739.55,A -85,B 0,C 180,E1 -17347.734,E2 -17347.734} C_VEL
LIN {X 0,Y 280.409,Z 748.914,A -85,B 0,C 180,E1 -17350.223,E2 -17350.223} C_VEL
LIN {X 0,Y 278.613,Z 756.701,A -85,B 0,C 180,E1 -17352.758,E2 -17352.758} C_VEL
LIN {X 0,Y 277.198,Z 763.141,A -85,B 0,C 180,E1 -17355.312,E2 -17355.312} C_VEL
LIN {X 0,Y 276.076,Z 769.044,A -85,B 0,C 180,E1 -17358.249,E2 -17358.249} C_VEL
LIN {X 0,Y 275.504,Z 773.559,A -85,B 0,C 180,E1 -17361.195,E2 -17361.195} C_VEL
LIN {X 0,Y 275.274,Z 776.787,A -85,B 0,C 180,E1 -17364.138,E2 -17364.138} C_VEL
LIN {X 0,Y 275.232,Z 778.745,A -85,B 0,C 180,E1 -17367.072,E2 -17367.072} C_VEL
LIN {X 0,Y 275.276,Z 779.517,A -85,B 0,C 180,E1 -17369.999,E2 -17369.999} C_VEL
LIN {X 0,Y 275.235,Z 779.131,A -85,B 0,C 180,E1 -17372.926,E2 -17372.926} C_VEL
LIN {X 0,Y 275.244,Z 777.595,A -85,B 0,C 180,E1 -17375.861,E2 -17375.861} C_VEL
LIN {X 0,Y 275.498,Z 774.886,A -85,B 0,C 180,E1 -17378.803,E2 -17378.803} C_VEL
LIN {X 0,Y 276.117,Z 770.908,A -85,B 0,C 180,E1 -17381.748,E2 -17381.748} C_VEL
LIN {X 0,Y 277.263,Z 765.61,A -85,B 0,C 180,E1 -17384.682,E2 -17384.682} C_VEL
LIN {X 0,Y 278.944,Z 758.883,A -85,B 0,C 180,E1 -17387.597,E2 -17387.597} C_VEL
LIN {X 0,Y 280.955,Z 751.662,A -85,B 0,C 180,E1 -17390.117,E2 -17390.117} C_VEL
LIN {X 0,Y 283.545,Z 743.018,A -85,B 0,C 180,E1 -17392.592,E2 -17392.592} C_VEL
LIN {X 0,Y 286.418,Z 732.646,A -85,B 0,C 180,E1 -17395.04,E2 -17395.04} C_VEL
LIN {X 0,Y 289.372,Z 722.053,A -85,B 0,C 180,E1 -17397.088,E2 -17397.088} C_VEL
LIN {X 0,Y 292.452,Z 710.554,A -85,B 0,C 180,E1 -17398.921,E2 -17398.921} C_VEL
LIN {X 0,Y 295.479,Z 698.095,A -85,B 0,C 180,E1 -17400.557,E2 -17400.557} C_VEL
LIN {X 0,Y 298.185,Z 685.557,A -85,B 0,C 180,E1 -17401.9,E2 -17401.9} C_VEL
LIN {X 0,Y 300.974,Z 670.453,A -85,B 0,C 180,E1 -17403.18,E2 -17403.18} C_VEL
LIN {X 0,Y 303.191,Z 656.074,A -85,B 0,C 180,E1 -17404.101,E2 -17404.101} C_VEL
LIN {X 0,Y 305.071,Z 640.465,A -85,B 0,C 180,E1 -17404.811,E2 -17404.811} C_VEL
LIN {X 0,Y 306.164,Z 625.329,A -85,B 0,C 180,E1 -17405.271,E2 -17405.271} C_VEL
LIN {X 0,Y 310.732,Z 526.352,A -85,B 0,C 180,E1 -17407.607,E2 -17407.607} C_VEL
LIN {X 0,Y 309.919,Z 520.797,A -85,B 0,C 180,E1 -17407.908,E2 -17407.908} C_VEL
LIN {X 0,Y 302.576,Z 504.165,A -85,B 0,C 180,E1 -17409.673,E2 -17409.673} C_VEL
LIN {X 0,Y 296.742,Z 492.787,A -85,B 0,C 180,E1 -17411.128,E2 -17411.128} C_VEL
LIN {X 0,Y 290.236,Z 481.104,A -85,B 0,C 180,E1 -17412.842,E2 -17412.842} C_VEL
LIN {X 0,Y 286.224,Z 474.721,A -85,B 0,C 180,E1 -17413.95,E2 -17413.95} C_VEL
LIN {X 0,Y 283.155,Z 470,A -85,B 0,C 180,E1 -17414.83,E2 -17414.83} C_VEL
LIN {X 0,Y 280.378,Z 465.649,A -85,B 0,C 180,E1 -17415.676,E2 -17415.676} C_VEL
LIN {X 0,Y 280.126,Z 464.924,A -85,B 0,C 180,E1 -17415.877,E2 -17415.877} C_VEL
LIN {X 0,Y 277.27,Z 456.57,A -85,B 0,C 180,E1 -17419.85,E2 -17419.85} C_VEL
LIN {X 0,Y 277.279,Z 456.566,A -85,B 0,C 180,E1 -17424.341,E2 -17424.341} C_VEL
LIN {X 0,Y 277.238,Z 456.573,A -85,B 0,C 180,E1 -17427.836,E2 -17427.836} C_VEL
LIN {X 0,Y 277.28,Z 456.572,A -85,B 0,C 180,E1 -17431.212,E2 -17431.212} C_VEL
LIN {X 0,Y 277.306,Z 456.569,A -85,B 0,C 180,E1 -17434.479,E2 -17434.479} C_VEL
LIN {X 0,Y 277.279,Z 456.571,A -85,B 0,C 180,E1 -17437.655,E2 -17437.655} C_VEL
LIN {X 0,Y 277.339,Z 456.561,A -85,B 0,C 180,E1 -17440.766,E2 -17440.766} C_VEL
LIN {X 0,Y 277.428,Z 456.552,A -85,B 0,C 180,E1 -17445.326,E2 -17445.326} C_VEL
LIN {X 0,Y 277.501,Z 456.536,A -85,B 0,C 180,E1 -17449.789,E2 -17449.789} C_VEL
LIN {X 0,Y 277.647,Z 456.524,A -85,B 0,C 180,E1 -17452.729,E2 -17452.729} C_VEL
LIN {X 0,Y 277.815,Z 456.498,A -85,B 0,C 180,E1 -17458.551,E2 -17458.551} C_VEL
LIN {X 0,Y 277.816,Z 456.494,A -85,B 0,C 180,E1 -17461.45,E2 -17461.45} C_VEL
LIN {X 0,Y 277.647,Z 456.521,A -85,B 0,C 180,E1 -17467.271,E2 -17467.271} C_VEL
LIN {X 0,Y 277.501,Z 456.541,A -85,B 0,C 180,E1 -17470.212,E2 -17470.212} C_VEL
LIN {X 0,Y 277.429,Z 456.549,A -85,B 0,C 180,E1 -17474.675,E2 -17474.675} C_VEL
LIN {X 0,Y 277.34,Z 456.56,A -85,B 0,C 180,E1 -17479.235,E2 -17479.235} C_VEL
LIN {X 0,Y 277.29,Z 456.569,A -85,B 0,C 180,E1 -17481.611,E2 -17481.611} C_VEL
LIN {X 0,Y 278.089,Z 459.102,A -85,B 0,C 180,E1 -17481.936,E2 -17481.936} C_VEL
LIN {X 0,Y 279.993,Z 461.296,A -85,B 0,C 180,E1 -17482.507,E2 -17482.507} C_VEL
LIN {X 0,Y 280.92,Z 462.084,A -85,B 0,C 180,E1 -17482.768,E2 -17482.768} C_VEL
LIN {X 0,Y 283.015,Z 465.455,A -85,B 0,C 180,E1 -17483.411,E2 -17483.411} C_VEL
LIN {X 0,Y 284.545,Z 467.215,A -85,B 0,C 180,E1 -17483.838,E2 -17483.838} C_VEL
LIN {X 0,Y 291.322,Z 476.969,A -85,B 0,C 180,E1 -17485.689,E2 -17485.689} C_VEL
LIN {X 0,Y 298.698,Z 489.351,A -85,B 0,C 180,E1 -17487.581,E2 -17487.581} C_VEL
LIN {X 0,Y 306.272,Z 503.825,A -85,B 0,C 180,E1 -17489.409,E2 -17489.409} C_VEL
LIN {X 0,Y 311.142,Z 514.685,A -85,B 0,C 180,E1 -17490.554,E2 -17490.554} C_VEL
LIN {X 0,Y 306.192,Z 619.527,A -85,B 0,C 180,E1 -17493.061,E2 -17493.061} C_VEL
LIN {X 0,Y 304.696,Z 635.314,A -85,B 0,C 180,E1 -17493.677,E2 -17493.677} C_VEL
LIN {X 0,Y 302.839,Z 650.14,A -85,B 0,C 180,E1 -17494.53,E2 -17494.53} C_VEL
LIN {X 0,Y 300.585,Z 664.503,A -85,B 0,C 180,E1 -17495.638,E2 -17495.638} C_VEL
LIN {X 0,Y 297.928,Z 678.068,A -85,B 0,C 180,E1 -17496.958,E2 -17496.958} C_VEL
LIN {X 0,Y 295.067,Z 690.551,A -85,B 0,C 180,E1 -17498.463,E2 -17498.463} C_VEL
LIN {X 0,Y 292.027,Z 702.843,A -85,B 0,C 180,E1 -17500.293,E2 -17500.293} C_VEL
LIN {X 0,Y 288.881,Z 714.258,A -85,B 0,C 180,E1 -17502.358,E2 -17502.358} C_VEL
LIN {X 0,Y 286.011,Z 724.208,A -85,B 0,C 180,E1 -17504.555,E2 -17504.555} C_VEL
LIN {X 0,Y 283.28,Z 733.267,A -85,B 0,C 180,E1 -17506.981,E2 -17506.981} C_VEL
LIN {X 0,Y 280.7,Z 741.947,A -85,B 0,C 180,E1 -17509.857,E2 -17509.857} C_VEL
LIN {X 0,Y 278.67,Z 748.87,A -85,B 0,C 180,E1 -17512.753,E2 -17512.753} C_VEL
LIN {X 0,Y 277.349,Z 753.58,A -85,B 0,C 180,E1 -17515.241,E2 -17515.241} C_VEL
LIN {X 0,Y 276.456,Z 757.344,A -85,B 0,C 180,E1 -17517.735,E2 -17517.735} C_VEL
LIN {X 0,Y 275.552,Z 760.863,A -85,B 0,C 180,E1 -17521.015,E2 -17521.015} C_VEL
LIN {X 0,Y 275.067,Z 762.892,A -85,B 0,C 180,E1 -17524.257,E2 -17524.257} C_VEL
LIN {X 0,Y 274.904,Z 763.529,A -85,B 0,C 180,E1 -17527.452,E2 -17527.452} C_VEL
LIN {X 0,Y 275.031,Z 762.829,A -85,B 0,C 180,E1 -17530.599,E2 -17530.599} C_VEL
LIN {X 0,Y 275.297,Z 760.849,A -85,B 0,C 180,E1 -17533.692,E2 -17533.692} C_VEL
LIN {X 0,Y 275.881,Z 757.59,A -85,B 0,C 180,E1 -17536.747,E2 -17536.747} C_VEL
LIN {X 0,Y 276.751,Z 753.025,A -85,B 0,C 180,E1 -17539.761,E2 -17539.761} C_VEL
LIN {X 0,Y 278.084,Z 747.054,A -85,B 0,C 180,E1 -17542.741,E2 -17542.741} C_VEL
LIN {X 0,Y 279.918,Z 739.522,A -85,B 0,C 180,E1 -17545.681,E2 -17545.681} C_VEL
LIN {X 0,Y 281.904,Z 731.487,A -85,B 0,C 180,E1 -17548.207,E2 -17548.207} C_VEL
LIN {X 0,Y 284.386,Z 721.765,A -85,B 0,C 180,E1 -17550.709,E2 -17550.709} C_VEL
LIN {X 0,Y 286.83,Z 711.875,A -85,B 0,C 180,E1 -17552.81,E2 -17552.81} C_VEL
LIN {X 0,Y 289.711,Z 699.724,A -85,B 0,C 180,E1 -17554.933,E2 -17554.933} C_VEL
LIN {X 0,Y 292.499,Z 687.096,A -85,B 0,C 180,E1 -17556.727,E2 -17556.727} C_VEL
LIN {X 0,Y 295.006,Z 674.227,A -85,B 0,C 180,E1 -17558.219,E2 -17558.219} C_VEL
LIN {X 0,Y 297.263,Z 660.234,A -85,B 0,C 180,E1 -17559.527,E2 -17559.527} C_VEL
LIN {X 0,Y 299.245,Z 645.731,A -85,B 0,C 180,E1 -17560.573,E2 -17560.573} C_VEL
LIN {X 0,Y 300.875,Z 629.98,A -85,B 0,C 180,E1 -17561.411,E2 -17561.411} C_VEL
LIN {X 0,Y 301.97,Z 614.595,A -85,B 0,C 180,E1 -17561.954,E2 -17561.954} C_VEL
LIN {X 0,Y 306.31,Z 512.136,A -85,B 0,C 180,E1 -17564.365,E2 -17564.365} C_VEL
LIN {X 0,Y 305.688,Z 509.825,A -85,B 0,C 180,E1 -17564.51,E2 -17564.51} C_VEL
LIN {X 0,Y 297.148,Z 491.407,A -85,B 0,C 180,E1 -17566.189,E2 -17566.189} C_VEL
LIN {X 0,Y 289.99,Z 477.615,A -85,B 0,C 180,E1 -17567.645,E2 -17567.645} C_VEL
LIN {X 0,Y 281.774,Z 464.48,A -85,B 0,C 180,E1 -17569.342,E2 -17569.342} C_VEL
LIN {X 0,Y 279.274,Z 460.573,A -85,B 0,C 180,E1 -17569.883,E2 -17569.883} C_VEL
LIN {X 0,Y 277.744,Z 458.169,A -85,B 0,C 180,E1 -17570.222,E2 -17570.222} C_VEL
LIN {X 0,Y 277.333,Z 456.561,A -85,B 0,C 180,E1 -17570.367,E2 -17570.367} C_VEL
LIN {X 0,Y 277.323,Z 456.556,A -85,B 0,C 180,E1 -17574.171,E2 -17574.171} C_VEL
LIN {X 0,Y 277.33,Z 456.555,A -85,B 0,C 180,E1 -17577.505,E2 -17577.505} C_VEL
LIN {X 0,Y 277.276,Z 456.573,A -85,B 0,C 180,E1 -17580.481,E2 -17580.481} C_VEL
LIN {X 0,Y 277.251,Z 456.566,A -85,B 0,C 180,E1 -17583.896,E2 -17583.896} C_VEL
LIN {X 0,Y 277.271,Z 456.555,A -85,B 0,C 180,E1 -17587.469,E2 -17587.469} C_VEL
LIN {X 0,Y 277.23,Z 456.578,A -85,B 0,C 180,E1 -17591.233,E2 -17591.233} C_VEL
LIN {X 0,Y 277.21,Z 456.578,A -85,B 0,C 180,E1 -17595.225,E2 -17595.225} C_VEL
LIN {X 0,Y 277.261,Z 456.562,A -85,B 0,C 180,E1 -17599.448,E2 -17599.448} C_VEL
LIN {X 0,Y 276.64,Z 456.651,A -85,B 0,C 180,E1 -17600.661,E2 -17600.661} C_VEL
LIN {X 0,Y 273.775,Z 457.002,A -85,B 0,C 180,E1 -17602.638,E2 -17602.638} C_VEL
LIN {X 0,Y 271.322,Z 457.301,A -85,B 0,C 180,E1 -17604.244,E2 -17604.244} C_VEL
LIN {X 0,Y 270.282,Z 457.433,A -85,B 0,C 180,E1 -17605.49,E2 -17605.49} C_VEL
LIN {X 0,Y 270.207,Z 457.446,A -85,B 0,C 180,E1 -17605.913,E2 -17605.913} C_VEL
LIN {X 0,Y 270.198,Z 457.434,A -85,B 0,C 180,E1 -17610.382,E2 -17610.382} C_VEL
LIN {X 0,Y 270.263,Z 457.445,A -85,B 0,C 180,E1 -17613.763,E2 -17613.763} C_VEL
LIN {X 0,Y 270.212,Z 457.429,A -85,B 0,C 180,E1 -17617.036,E2 -17617.036} C_VEL
LIN {X 0,Y 270.303,Z 457.438,A -85,B 0,C 180,E1 -17620.244,E2 -17620.244} C_VEL
LIN {X 0,Y 270.405,Z 457.416,A -85,B 0,C 180,E1 -17624.935,E2 -17624.935} C_VEL
LIN {X 0,Y 270.444,Z 457.403,A -85,B 0,C 180,E1 -17629.519,E2 -17629.519} C_VEL
LIN {X 0,Y 270.613,Z 457.398,A -85,B 0,C 180,E1 -17632.538,E2 -17632.538} C_VEL
LIN {X 0,Y 270.788,Z 457.368,A -85,B 0,C 180,E1 -17638.512,E2 -17638.512} C_VEL
LIN {X 0,Y 270.788,Z 457.377,A -85,B 0,C 180,E1 -17641.487,E2 -17641.487} C_VEL
LIN {X 0,Y 270.612,Z 457.397,A -85,B 0,C 180,E1 -17647.461,E2 -17647.461} C_VEL
LIN {X 0,Y 270.443,Z 457.409,A -85,B 0,C 180,E1 -17650.481,E2 -17650.481} C_VEL
LIN {X 0,Y 270.404,Z 457.426,A -85,B 0,C 180,E1 -17655.064,E2 -17655.064} C_VEL
LIN {X 0,Y 270.303,Z 457.425,A -85,B 0,C 180,E1 -17659.755,E2 -17659.755} C_VEL
LIN {X 0,Y 270.275,Z 457.443,A -85,B 0,C 180,E1 -17664.585,E2 -17664.585} C_VEL
LIN {X 0,Y 270.271,Z 457.441,A -85,B 0,C 180,E1 -17667.908,E2 -17667.908} C_VEL
LIN {X 0,Y 270.185,Z 457.451,A -85,B 0,C 180,E1 -17671.348,E2 -17671.348} C_VEL
LIN {X 0,Y 270.215,Z 457.451,A -85,B 0,C 180,E1 -17674.903,E2 -17674.903} C_VEL
LIN {X 0,Y 270.223,Z 457.449,A -85,B 0,C 180,E1 -17678.717,E2 -17678.717} C_VEL
LIN {X 0,Y 270.195,Z 457.451,A -85,B 0,C 180,E1 -17682.553,E2 -17682.553} C_VEL
LIN {X 0,Y 270.225,Z 457.611,A -85,B 0,C 180,E1 -17683.495,E2 -17683.495} C_VEL
LIN {X 0,Y 273.012,Z 466.629,A -85,B 0,C 180,E1 -17686.856,E2 -17686.856} C_VEL
LIN {X 0,Y 275.604,Z 471.167,A -85,B 0,C 180,E1 -17687.455,E2 -17687.455} C_VEL
LIN {X 0,Y 285.654,Z 490.271,A -85,B 0,C 180,E1 -17689.702,E2 -17689.702} C_VEL
LIN {X 0,Y 293.803,Z 507.635,A -85,B 0,C 180,E1 -17691.435,E2 -17691.435} C_VEL
LIN {X 0,Y 299.11,Z 520.08,A -85,B 0,C 180,E1 -17692.535,E2 -17692.535} C_VEL
LIN {X 0,Y 299.979,Z 527.097,A -85,B 0,C 180,E1 -17692.858,E2 -17692.858} C_VEL
LIN {X 0,Y 295.379,Z 633.561,A -85,B 0,C 180,E1 -17695.436,E2 -17695.436} C_VEL
LIN {X 0,Y 293.944,Z 649.598,A -85,B 0,C 180,E1 -17696.073,E2 -17696.073} C_VEL
LIN {X 0,Y 291.885,Z 665.406,A -85,B 0,C 180,E1 -17696.991,E2 -17696.991} C_VEL
LIN {X 0,Y 289.767,Z 678.761,A -85,B 0,C 180,E1 -17698.024,E2 -17698.024} C_VEL
LIN {X 0,Y 287.04,Z 693.274,A -85,B 0,C 180,E1 -17699.465,E2 -17699.465} C_VEL
LIN {X 0,Y 284.052,Z 706.802,A -85,B 0,C 180,E1 -17701.153,E2 -17701.153} C_VEL
LIN {X 0,Y 281.136,Z 719.125,A -85,B 0,C 180,E1 -17703.057,E2 -17703.057} C_VEL
LIN {X 0,Y 278.524,Z 729.521,A -85,B 0,C 180,E1 -17705.001,E2 -17705.001} C_VEL
LIN {X 0,Y 275.845,Z 740.592,A -85,B 0,C 180,E1 -17707.531,E2 -17707.531} C_VEL
LIN {X 0,Y 273.349,Z 749.753,A -85,B 0,C 180,E1 -17710.082,E2 -17710.082} C_VEL
LIN {X 0,Y 271.51,Z 757.354,A -85,B 0,C 180,E1 -17712.681,E2 -17712.681} C_VEL
LIN {X 0,Y 269.907,Z 764.44,A -85,B 0,C 180,E1 -17715.678,E2 -17715.678} C_VEL
LIN {X 0,Y 268.852,Z 769.999,A -85,B 0,C 180,E1 -17718.693,E2 -17718.693} C_VEL
LIN {X 0,Y 268.443,Z 773.282,A -85,B 0,C 180,E1 -17720.962,E2 -17720.962} C_VEL
LIN {X 0,Y 268.204,Z 776.531,A -85,B 0,C 180,E1 -17723.983,E2 -17723.983} C_VEL
LIN {X 0,Y 268.144,Z 778.507,A -85,B 0,C 180,E1 -17726.994,E2 -17726.994} C_VEL
LIN {X 0,Y 268.2,Z 779.303,A -85,B 0,C 180,E1 -17729.999,E2 -17729.999} C_VEL
LIN {X 0,Y 268.146,Z 778.941,A -85,B 0,C 180,E1 -17733.004,E2 -17733.004} C_VEL
LIN {X 0,Y 268.154,Z 777.426,A -85,B 0,C 180,E1 -17736.017,E2 -17736.017} C_VEL
LIN {X 0,Y 268.44,Z 774.736,A -85,B 0,C 180,E1 -17739.037,E2 -17739.037} C_VEL
LIN {X 0,Y 269.112,Z 770.781,A -85,B 0,C 180,E1 -17742.058,E2 -17742.058} C_VEL
LIN {X 0,Y 270.341,Z 765.519,A -85,B 0,C 180,E1 -17745.067,E2 -17745.067} C_VEL
LIN {X 0,Y 272.122,Z 758.823,A -85,B 0,C 180,E1 -17748.053,E2 -17748.053} C_VEL
LIN {X 0,Y 274.249,Z 751.636,A -85,B 0,C 180,E1 -17750.631,E2 -17750.631} C_VEL
LIN {X 0,Y 276.951,Z 743.029,A -85,B 0,C 180,E1 -17753.161,E2 -17753.161} C_VEL
LIN {X 0,Y 279.94,Z 732.708,A -85,B 0,C 180,E1 -17755.661,E2 -17755.661} C_VEL
LIN {X 0,Y 283.059,Z 722.19,A -85,B 0,C 180,E1 -17757.744,E2 -17757.744} C_VEL
LIN {X 0,Y 286.262,Z 710.784,A -85,B 0,C 180,E1 -17759.608,E2 -17759.608} C_VEL
LIN {X 0,Y 289.386,Z 698.427,A -85,B 0,C 180,E1 -17761.271,E2 -17761.271} C_VEL
LIN {X 0,Y 292.476,Z 684.739,A -85,B 0,C 180,E1 -17762.752,E2 -17762.752} C_VEL
LIN {X 0,Y 295.085,Z 671.054,A -85,B 0,C 180,E1 -17763.931,E2 -17763.931} C_VEL
LIN {X 0,Y 297.58,Z 655.534,A -85,B 0,C 180,E1 -17764.939,E2 -17764.939} C_VEL
LIN {X 0,Y 299.528,Z 639.751,A -85,B 0,C 180,E1 -17765.655,E2 -17765.655} C_VEL
LIN {X 0,Y 300.628,Z 624.371,A -85,B 0,C 180,E1 -17766.124,E2 -17766.124} C_VEL
LIN {X 0,Y 304.91,Z 535.103,A -85,B 0,C 180,E1 -17768.269,E2 -17768.269} C_VEL
LIN {X 0,Y 305.276,Z 526.382,A -85,B 0,C 180,E1 -17768.488,E2 -17768.488} C_VEL
LIN {X 0,Y 304.682,Z 523.507,A -85,B 0,C 180,E1 -17768.68,E2 -17768.68} C_VEL
LIN {X 0,Y 297.268,Z 506.686,A -85,B 0,C 180,E1 -17770.546,E2 -17770.546} C_VEL
LIN {X 0,Y 290.138,Z 492.855,A -85,B 0,C 180,E1 -17772.43,E2 -17772.43} C_VEL
LIN {X 0,Y 284.664,Z 483.433,A -85,B 0,C 180,E1 -17773.959,E2 -17773.959} C_VEL
LIN {X 0,Y 279.745,Z 475.509,A -85,B 0,C 180,E1 -17775.423,E2 -17775.423} C_VEL
LIN {X 0,Y 275.773,Z 469.543,A -85,B 0,C 180,E1 -17776.671,E2 -17776.671} C_VEL
LIN {X 0,Y 272.74,Z 464.87,A -85,B 0,C 180,E1 -17777.686,E2 -17777.686} C_VEL
LIN {X 0,Y 270.203,Z 457.45,A -85,B 0,C 180,E1 -17781.493,E2 -17781.493} C_VEL
LIN {X 0,Y 270.196,Z 457.45,A -85,B 0,C 180,E1 -17785.094,E2 -17785.094} C_VEL
LIN {X 0,Y 270.194,Z 457.451,A -85,B 0,C 180,E1 -17789.13,E2 -17789.13} C_VEL
LIN {X 0,Y 270.258,Z 457.442,A -85,B 0,C 180,E1 -17792.146,E2 -17792.146} C_VEL
LIN {X 0,Y 270.271,Z 457.439,A -85,B 0,C 180,E1 -17795.519,E2 -17795.519} C_VEL
LIN {X 0,Y 270.295,Z 457.433,A -85,B 0,C 180,E1 -17800.244,E2 -17800.244} C_VEL
LIN {X 0,Y 270.397,Z 457.429,A -85,B 0,C 180,E1 -17804.935,E2 -17804.935} C_VEL
LIN {X 0,Y 270.436,Z 457.418,A -85,B 0,C 180,E1 -17809.519,E2 -17809.519} C_VEL
LIN {X 0,Y 270.605,Z 457.403,A -85,B 0,C 180,E1 -17812.539,E2 -17812.539} C_VEL
LIN {X 0,Y 270.781,Z 457.373,A -85,B 0,C 180,E1 -17818.513,E2 -17818.513} C_VEL
LIN {X 0,Y 270.781,Z 457.37,A -85,B 0,C 180,E1 -17821.488,E2 -17821.488} C_VEL
LIN {X 0,Y 270.605,Z 457.397,A -85,B 0,C 180,E1 -17827.462,E2 -17827.462} C_VEL
LIN {X 0,Y 270.436,Z 457.418,A -85,B 0,C 180,E1 -17830.482,E2 -17830.482} C_VEL
LIN {X 0,Y 270.397,Z 457.428,A -85,B 0,C 180,E1 -17835.065,E2 -17835.065} C_VEL
LIN {X 0,Y 270.3,Z 457.439,A -85,B 0,C 180,E1 -17839.756,E2 -17839.756} C_VEL
LIN {X 0,Y 271.185,Z 460.116,A -85,B 0,C 180,E1 -17840.141,E2 -17840.141} C_VEL
LIN {X 0,Y 273.149,Z 462.339,A -85,B 0,C 180,E1 -17840.78,E2 -17840.78} C_VEL
LIN {X 0,Y 274.003,Z 463.135,A -85,B 0,C 180,E1 -17841.045,E2 -17841.045} C_VEL
LIN {X 0,Y 276.021,Z 466.364,A -85,B 0,C 180,E1 -17841.716,E2 -17841.716} C_VEL
LIN {X 0,Y 277.807,Z 468.256,A -85,B 0,C 180,E1 -17842.252,E2 -17842.252} C_VEL
LIN {X 0,Y 280.429,Z 471.905,A -85,B 0,C 180,E1 -17843.054,E2 -17843.054} C_VEL
LIN {X 0,Y 287.023,Z 481.316,A -85,B 0,C 180,E1 -17844.937,E2 -17844.937} C_VEL
LIN {X 0,Y 293.639,Z 492.367,A -85,B 0,C 180,E1 -17846.713,E2 -17846.713} C_VEL
LIN {X 0,Y 301.539,Z 507.679,A -85,B 0,C 180,E1 -17848.719,E2 -17848.719} C_VEL
LIN {X 0,Y 305.669,Z 516.733,A -85,B 0,C 180,E1 -17849.724,E2 -17849.724} C_VEL
LIN {X 0,Y 300.645,Z 619.534,A -85,B 0,C 180,E1 -17852.23,E2 -17852.23} C_VEL
LIN {X 0,Y 299.069,Z 635.432,A -85,B 0,C 180,E1 -17852.851,E2 -17852.851} C_VEL
LIN {X 0,Y 297.218,Z 649.923,A -85,B 0,C 180,E1 -17853.693,E2 -17853.693} C_VEL
LIN {X 0,Y 294.827,Z 664.491,A -85,B 0,C 180,E1 -17854.821,E2 -17854.821} C_VEL
LIN {X 0,Y 291.912,Z 678.835,A -85,B 0,C 180,E1 -17856.243,E2 -17856.243} C_VEL
LIN {X 0,Y 288.896,Z 691.493,A -85,B 0,C 180,E1 -17857.805,E2 -17857.805} C_VEL
LIN {X 0,Y 285.538,Z 704.375,A -85,B 0,C 180,E1 -17859.788,E2 -17859.788} C_VEL
LIN {X 0,Y 282.512,Z 714.774,A -85,B 0,C 180,E1 -17861.731,E2 -17861.731} C_VEL
LIN {X 0,Y 279.272,Z 725.501,A -85,B 0,C 180,E1 -17864.177,E2 -17864.177} C_VEL
LIN {X 0,Y 276.437,Z 734.365,A -85,B 0,C 180,E1 -17866.653,E2 -17866.653} C_VEL
LIN {X 0,Y 273.773,Z 742.879,A -85,B 0,C 180,E1 -17869.596,E2 -17869.596} C_VEL
LIN {X 0,Y 271.67,Z 749.657,A -85,B 0,C 180,E1 -17872.561,E2 -17872.561} C_VEL
LIN {X 0,Y 269.99,Z 755.432,A -85,B 0,C 180,E1 -17875.862,E2 -17875.862} C_VEL
LIN {X 0,Y 269.114,Z 758.856,A -85,B 0,C 180,E1 -17878.514,E2 -17878.514} C_VEL
LIN {X 0,Y 268.293,Z 761.873,A -85,B 0,C 180,E1 -17881.869,E2 -17881.869} C_VEL
LIN {X 0,Y 267.862,Z 763.431,A -85,B 0,C 180,E1 -17885.179,E2 -17885.179} C_VEL
LIN {X 0,Y 267.769,Z 763.62,A -85,B 0,C 180,E1 -17888.443,E2 -17888.443} C_VEL
LIN {X 0,Y 268.002,Z 762.497,A -85,B 0,C 180,E1 -17891.659,E2 -17891.659} C_VEL
LIN {X 0,Y 268.372,Z 760.11,A -85,B 0,C 180,E1 -17894.82,E2 -17894.82} C_VEL
LIN {X 0,Y 269.098,Z 756.434,A -85,B 0,C 180,E1 -17897.941,E2 -17897.941} C_VEL
LIN {X 0,Y 270.232,Z 751.045,A -85,B 0,C 180,E1 -17901.221,E2 -17901.221} C_VEL
LIN {X 0,Y 271.681,Z 744.968,A -85,B 0,C 180,E1 -17904.062,E2 -17904.062} C_VEL
LIN {X 0,Y 273.799,Z 736.855,A -85,B 0,C 180,E1 -17907.058,E2 -17907.058} C_VEL
LIN {X 0,Y 276.09,Z 728.206,A -85,B 0,C 180,E1 -17909.636,E2 -17909.636} C_VEL
LIN {X 0,Y 278.853,Z 717.787,A -85,B 0,C 180,E1 -17912.167,E2 -17912.167} C_VEL
LIN {X 0,Y 281.522,Z 707.134,A -85,B 0,C 180,E1 -17914.296,E2 -17914.296} C_VEL
LIN {X 0,Y 284.266,Z 695.526,A -85,B 0,C 180,E1 -17916.21,E2 -17916.21} C_VEL
LIN {X 0,Y 287.055,Z 682.861,A -85,B 0,C 180,E1 -17917.916,E2 -17917.916} C_VEL
LIN {X 0,Y 289.707,Z 668.983,A -85,B 0,C 180,E1 -17919.425,E2 -17919.425} C_VEL
LIN {X 0,Y 291.838,Z 655.675,A -85,B 0,C 180,E1 -17920.582,E2 -17920.582} C_VEL
LIN {X 0,Y 293.662,Z 641.791,A -85,B 0,C 180,E1 -17921.519,E2 -17921.519} C_VEL
LIN {X 0,Y 295.188,Z 626.361,A -85,B 0,C 180,E1 -17922.278,E2 -17922.278} C_VEL
LIN {X 0,Y 296.196,Z 609.706,A -85,B 0,C 180,E1 -17922.801,E2 -17922.801} C_VEL
LIN {X 0,Y 300.31,Z 513.27,A -85,B 0,C 180,E1 -17925.106,E2 -17925.106} C_VEL
LIN {X 0,Y 292.209,Z 495.528,A -85,B 0,C 180,E1 -17926.763,E2 -17926.763} C_VEL
LIN {X 0,Y 285.257,Z 482.105,A -85,B 0,C 180,E1 -17928.215,E2 -17928.215} C_VEL
LIN {X 0,Y 277.233,Z 469.157,A -85,B 0,C 180,E1 -17929.933,E2 -17929.933} C_VEL
LIN {X 0,Y 274.502,Z 464.997,A -85,B 0,C 180,E1 -17930.538,E2 -17930.538} C_VEL
LIN {X 0,Y 272.423,Z 461.739,A -85,B 0,C 180,E1 -17931.011,E2 -17931.011} C_VEL
LIN {X 0,Y 270.692,Z 459.188,A -85,B 0,C 180,E1 -17931.406,E2 -17931.406} C_VEL
LIN {X 0,Y 270.229,Z 457.444,A -85,B 0,C 180,E1 -17931.554,E2 -17931.554} C_VEL
LIN {X 0,Y 270.278,Z 457.433,A -85,B 0,C 180,E1 -17934.586,E2 -17934.586} C_VEL
LIN {X 0,Y 270.274,Z 457.431,A -85,B 0,C 180,E1 -17937.909,E2 -17937.909} C_VEL
LIN {X 0,Y 270.188,Z 457.447,A -85,B 0,C 180,E1 -17941.348,E2 -17941.348} C_VEL
LIN {X 0,Y 270.206,Z 457.453,A -85,B 0,C 180,E1 -17944.905,E2 -17944.905} C_VEL
LIN {X 0,Y 270.226,Z 457.433,A -85,B 0,C 180,E1 -17948.717,E2 -17948.717} C_VEL
LIN {X 0,Y 270.182,Z 457.445,A -85,B 0,C 180,E1 -17952.557,E2 -17952.557} C_VEL
LIN {X 0,Y 270.183,Z 457.453,A -85,B 0,C 180,E1 -17956.747,E2 -17956.747} C_VEL
LIN {X 0,Y 270.215,Z 457.44,A -85,B 0,C 180,E1 -17959.441,E2 -17959.441} C_VEL
LIN {X 0,Y 270.243,Z 457.434,A -85,B 0,C 180,E1 -17963.262,E2 -17963.262} C_VEL
LIN {X 0,Y 270.207,Z 457.446,A -85,B 0,C 180,E1 -17965.913,E2 -17965.913} C_VEL
LIN {X 0,Y 269.562,Z 457.534,A -85,B 0,C 180,E1 -17967.156,E2 -17967.156} C_VEL
LIN {X 0,Y 266.716,Z 457.884,A -85,B 0,C 180,E1 -17969.181,E2 -17969.181} C_VEL
LIN {X 0,Y 264.292,Z 458.179,A -85,B 0,C 180,E1 -17970.828,E2 -17970.828} C_VEL
LIN {X 0,Y 263.26,Z 458.312,A -85,B 0,C 180,E1 -17972.105,E2 -17972.105} C_VEL
LIN {X 0,Y 263.181,Z 458.321,A -85,B 0,C 180,E1 -17972.537,E2 -17972.537} C_VEL
LIN {X 0,Y 263.157,Z 458.307,A -85,B 0,C 180,E1 -17976.384,E2 -17976.384} C_VEL
LIN {X 0,Y 263.265,Z 458.317,A -85,B 0,C 180,E1 -17979.693,E2 -17979.693} C_VEL
LIN {X 0,Y 263.353,Z 458.289,A -85,B 0,C 180,E1 -17984.522,E2 -17984.522} C_VEL
LIN {X 0,Y 263.376,Z 458.285,A -85,B 0,C 180,E1 -17989.234,E2 -17989.234} C_VEL
LIN {X 0,Y 263.574,Z 458.272,A -85,B 0,C 180,E1 -17992.338,E2 -17992.338} C_VEL
LIN {X 0,Y 263.752,Z 458.243,A -85,B 0,C 180,E1 -17998.473,E2 -17998.473} C_VEL
LIN {X 0,Y 263.753,Z 458.253,A -85,B 0,C 180,E1 -18001.527,E2 -18001.527} C_VEL
LIN {X 0,Y 263.574,Z 458.276,A -85,B 0,C 180,E1 -18007.661,E2 -18007.661} C_VEL
LIN {X 0,Y 263.375,Z 458.285,A -85,B 0,C 180,E1 -18010.765,E2 -18010.765} C_VEL
LIN {X 0,Y 263.352,Z 458.307,A -85,B 0,C 180,E1 -18015.478,E2 -18015.478} C_VEL
LIN {X 0,Y 263.269,Z 458.307,A -85,B 0,C 180,E1 -18020.306,E2 -18020.306} C_VEL
LIN {X 0,Y 263.21,Z 458.322,A -85,B 0,C 180,E1 -18025.291,E2 -18025.291} C_VEL
LIN {X 0,Y 263.177,Z 458.324,A -85,B 0,C 180,E1 -18028.729,E2 -18028.729} C_VEL
LIN {X 0,Y 263.134,Z 458.333,A -85,B 0,C 180,E1 -18032.288,E2 -18032.288} C_VEL
LIN {X 0,Y 263.188,Z 458.323,A -85,B 0,C 180,E1 -18035.977,E2 -18035.977} C_VEL
LIN {X 0,Y 263.123,Z 458.332,A -85,B 0,C 180,E1 -18039.869,E2 -18039.869} C_VEL
LIN {X 0,Y 263.158,Z 458.378,A -85,B 0,C 180,E1 -18042.402,E2 -18042.402} C_VEL
LIN {X 0,Y 265.638,Z 466.396,A -85,B 0,C 180,E1 -18045.521,E2 -18045.521} C_VEL
LIN {X 0,Y 274.194,Z 481.672,A -85,B 0,C 180,E1 -18047.579,E2 -18047.579} C_VEL
LIN {X 0,Y 282.969,Z 498.954,A -85,B 0,C 180,E1 -18049.574,E2 -18049.574} C_VEL
LIN {X 0,Y 291.408,Z 517.79,A -85,B 0,C 180,E1 -18051.411,E2 -18051.411} C_VEL
LIN {X 0,Y 293.623,Z 523.43,A -85,B 0,C 180,E1 -18051.894,E2 -18051.894} C_VEL
LIN {X 0,Y 294.116,Z 527.774,A -85,B 0,C 180,E1 -18052.095,E2 -18052.095} C_VEL
LIN {X 0,Y 289.405,Z 632.607,A -85,B 0,C 180,E1 -18054.671,E2 -18054.671} C_VEL
LIN {X 0,Y 288.078,Z 648.112,A -85,B 0,C 180,E1 -18055.284,E2 -18055.284} C_VEL
LIN {X 0,Y 286.052,Z 663.081,A -85,B 0,C 180,E1 -18056.123,E2 -18056.123} C_VEL
LIN {X 0,Y 283.677,Z 678.021,A -85,B 0,C 180,E1 -18057.275,E2 -18057.275} C_VEL
LIN {X 0,Y 280.894,Z 692.507,A -85,B 0,C 180,E1 -18058.723,E2 -18058.723} C_VEL
LIN {X 0,Y 278.09,Z 704.876,A -85,B 0,C 180,E1 -18060.266,E2 -18060.266} C_VEL
LIN {X 0,Y 275.027,Z 717.491,A -85,B 0,C 180,E1 -18062.201,E2 -18062.201} C_VEL
LIN {X 0,Y 272.448,Z 727.146,A -85,B 0,C 180,E1 -18063.989,E2 -18063.989} C_VEL
LIN {X 0,Y 269.906,Z 737.096,A -85,B 0,C 180,E1 -18066.196,E2 -18066.196} C_VEL
LIN {X 0,Y 267.606,Z 745.572,A -85,B 0,C 180,E1 -18068.427,E2 -18068.427} C_VEL
LIN {X 0,Y 265.432,Z 753.885,A -85,B 0,C 180,E1 -18071.073,E2 -18071.073} C_VEL
LIN {X 0,Y 263.621,Z 761.016,A -85,B 0,C 180,E1 -18073.867,E2 -18073.867} C_VEL
LIN {X 0,Y 262.372,Z 767.073,A -85,B 0,C 180,E1 -18076.839,E2 -18076.839} C_VEL
LIN {X 0,Y 261.528,Z 771.965,A -85,B 0,C 180,E1 -18079.94,E2 -18079.94} C_VEL
LIN {X 0,Y 261.209,Z 774.799,A -85,B 0,C 180,E1 -18082.268,E2 -18082.268} C_VEL
LIN {X 0,Y 261.017,Z 777.418,A -85,B 0,C 180,E1 -18085.366,E2 -18085.366} C_VEL
LIN {X 0,Y 261.108,Z 778.825,A -85,B 0,C 180,E1 -18088.457,E2 -18088.457} C_VEL
LIN {X 0,Y 261.109,Z 779.065,A -85,B 0,C 180,E1 -18091.541,E2 -18091.541} C_VEL
LIN {X 0,Y 261.016,Z 778.151,A -85,B 0,C 180,E1 -18094.632,E2 -18094.632} C_VEL
LIN {X 0,Y 261.207,Z 776.084,A -85,B 0,C 180,E1 -18097.73,E2 -18097.73} C_VEL
LIN {X 0,Y 261.716,Z 772.783,A -85,B 0,C 180,E1 -18100.834,E2 -18100.834} C_VEL
LIN {X 0,Y 262.754,Z 768.215,A -85,B 0,C 180,E1 -18103.928,E2 -18103.928} C_VEL
LIN {X 0,Y 264.262,Z 762.283,A -85,B 0,C 180,E1 -18107.009,E2 -18107.009} C_VEL
LIN {X 0,Y 266.55,Z 754.841,A -85,B 0,C 180,E1 -18110.044,E2 -18110.044} C_VEL
LIN {X 0,Y 269.115,Z 746.917,A -85,B 0,C 180,E1 -18112.655,E2 -18112.655} C_VEL
LIN {X 0,Y 271.884,Z 738.059,A -85,B 0,C 180,E1 -18115.073,E2 -18115.073} C_VEL
LIN {X 0,Y 275.075,Z 727.802,A -85,B 0,C 180,E1 -18117.379,E2 -18117.379} C_VEL
LIN {X 0,Y 278.506,Z 716.4,A -85,B 0,C 180,E1 -18119.476,E2 -18119.476} C_VEL
LIN {X 0,Y 281.984,Z 703.891,A -85,B 0,C 180,E1 -18121.349,E2 -18121.349} C_VEL
LIN {X 0,Y 285.365,Z 690.518,A -85,B 0,C 180,E1 -18122.956,E2 -18122.956} C_VEL
LIN {X 0,Y 288.313,Z 676.538,A -85,B 0,C 180,E1 -18124.311,E2 -18124.311} C_VEL
LIN {X 0,Y 291.024,Z 661.555,A -85,B 0,C 180,E1 -18125.42,E2 -18125.42} C_VEL
LIN {X 0,Y 293.213,Z 646.601,A -85,B 0,C 180,E1 -18126.225,E2 -18126.225} C_VEL
LIN {X 0,Y 294.696,Z 631.161,A -85,B 0,C 180,E1 -18126.81,E2 -18126.81} C_VEL
LIN {X 0,Y 299.313,Z 541.437,A -85,B 0,C 180,E1 -18129.009,E2 -18129.009} C_VEL
LIN {X 0,Y 299.953,Z 527.534,A -85,B 0,C 180,E1 -18129.358,E2 -18129.358} C_VEL
LIN {X 0,Y 293.55,Z 512.476,A -85,B 0,C 180,E1 -18131.049,E2 -18131.049} C_VEL
LIN {X 0,Y 286.989,Z 499.282,A -85,B 0,C 180,E1 -18132.848,E2 -18132.848} C_VEL
LIN {X 0,Y 281.374,Z 489.311,A -85,B 0,C 180,E1 -18134.476,E2 -18134.476} C_VEL
LIN {X 0,Y 276.288,Z 480.873,A -85,B 0,C 180,E1 -18136.056,E2 -18136.056} C_VEL
LIN {X 0,Y 271.944,Z 474.382,A -85,B 0,C 180,E1 -18137.471,E2 -18137.471} C_VEL
LIN {X 0,Y 268.844,Z 469.796,A -85,B 0,C 180,E1 -18138.536,E2 -18138.536} C_VEL
LIN {X 0,Y 265.534,Z 464.918,A -85,B 0,C 180,E1 -18139.763,E2 -18139.763} C_VEL
LIN {X 0,Y 264.997,Z 463.742,A -85,B 0,C 180,E1 -18140.272,E2 -18140.272} C_VEL
LIN {X 0,Y 263.167,Z 458.33,A -85,B 0,C 180,E1 -18143.366,E2 -18143.366} C_VEL
LIN {X 0,Y 263.162,Z 458.331,A -85,B 0,C 180,E1 -18145.887,E2 -18145.887} C_VEL
LIN {X 0,Y 263.144,Z 458.326,A -85,B 0,C 180,E1 -18149.506,E2 -18149.506} C_VEL
LIN {X 0,Y 263.185,Z 458.319,A -85,B 0,C 180,E1 -18153.002,E2 -18153.002} C_VEL
LIN {X 0,Y 263.177,Z 458.319,A -85,B 0,C 180,E1 -18156.387,E2 -18156.387} C_VEL
LIN {X 0,Y 263.257,Z 458.308,A -85,B 0,C 180,E1 -18159.693,E2 -18159.693} C_VEL
LIN {X 0,Y 263.345,Z 458.305,A -85,B 0,C 180,E1 -18164.522,E2 -18164.522} C_VEL
LIN {X 0,Y 263.368,Z 458.301,A -85,B 0,C 180,E1 -18169.235,E2 -18169.235} C_VEL
LIN {X 0,Y 263.566,Z 458.281,A -85,B 0,C 180,E1 -18172.339,E2 -18172.339} C_VEL
LIN {X 0,Y 263.746,Z 458.249,A -85,B 0,C 180,E1 -18178.473,E2 -18178.473} C_VEL
LIN {X 0,Y 263.746,Z 458.247,A -85,B 0,C 180,E1 -18181.527,E2 -18181.527} C_VEL
LIN {X 0,Y 263.567,Z 458.272,A -85,B 0,C 180,E1 -18187.662,E2 -18187.662} C_VEL
LIN {X 0,Y 263.368,Z 458.297,A -85,B 0,C 180,E1 -18190.766,E2 -18190.766} C_VEL
LIN {X 0,Y 263.345,Z 458.308,A -85,B 0,C 180,E1 -18195.479,E2 -18195.479} C_VEL
LIN {X 0,Y 263.247,Z 458.318,A -85,B 0,C 180,E1 -18197.629,E2 -18197.629} C_VEL
LIN {X 0,Y 264.044,Z 460.83,A -85,B 0,C 180,E1 -18198.025,E2 -18198.025} C_VEL
LIN {X 0,Y 266.079,Z 463.175,A -85,B 0,C 180,E1 -18198.779,E2 -18198.779} C_VEL
LIN {X 0,Y 267.164,Z 463.966,A -85,B 0,C 180,E1 -18199.149,E2 -18199.149} C_VEL
LIN {X 0,Y 269.136,Z 467.226,A -85,B 0,C 180,E1 -18199.886,E2 -18199.886} C_VEL
LIN {X 0,Y 271.056,Z 469.419,A -85,B 0,C 180,E1 -18200.525,E2 -18200.525} C_VEL
LIN {X 0,Y 273.871,Z 473.173,A -85,B 0,C 180,E1 -18201.45,E2 -18201.45} C_VEL
LIN {X 0,Y 278.573,Z 479.667,A -85,B 0,C 180,E1 -18202.922,E2 -18202.922} C_VEL
LIN {X 0,Y 284.845,Z 488.932,A -85,B 0,C 180,E1 -18204.751,E2 -18204.751} C_VEL
LIN {X 0,Y 291.75,Z 501.273,A -85,B 0,C 180,E1 -18206.658,E2 -18206.658} C_VEL
LIN {X 0,Y 298.547,Z 515.198,A -85,B 0,C 180,E1 -18208.438,E2 -18208.438} C_VEL
LIN {X 0,Y 300.337,Z 519.309,A -85,B 0,C 180,E1 -18208.894,E2 -18208.894} C_VEL
LIN {X 0,Y 295.157,Z 619.847,A -85,B 0,C 180,E1 -18211.368,E2 -18211.368} C_VEL
LIN {X 0,Y 293.504,Z 635.901,A -85,B 0,C 180,E1 -18212.007,E2 -18212.007} C_VEL
LIN {X 0,Y 291.441,Z 651.121,A -85,B 0,C 180,E1 -18212.916,E2 -18212.916} C_VEL
LIN {X 0,Y 289.1,Z 664.766,A -85,B 0,C 180,E1 -18213.996,E2 -18213.996} C_VEL
LIN {X 0,Y 286.329,Z 677.884,A -85,B 0,C 180,E1 -18215.303,E2 -18215.303} C_VEL
LIN {X 0,Y 283.026,Z 691.356,A -85,B 0,C 180,E1 -18216.971,E2 -18216.971} C_VEL
LIN {X 0,Y 279.589,Z 704.035,A -85,B 0,C 180,E1 -18218.934,E2 -18218.934} C_VEL
LIN {X 0,Y 276.197,Z 715.318,A -85,B 0,C 180,E1 -18221.079,E2 -18221.079} C_VEL
LIN {X 0,Y 273.075,Z 725.146,A -85,B 0,C 180,E1 -18223.362,E2 -18223.362} C_VEL
LIN {X 0,Y 270.061,Z 734.094,A -85,B 0,C 180,E1 -18225.885,E2 -18225.885} C_VEL
LIN {X 0,Y 267.581,Z 741.544,A -85,B 0,C 180,E1 -18228.458,E2 -18228.458} C_VEL
LIN {X 0,Y 265.218,Z 748.628,A -85,B 0,C 180,E1 -18231.486,E2 -18231.486} C_VEL
LIN {X 0,Y 263.674,Z 753.5,A -85,B 0,C 180,E1 -18234.1,E2 -18234.1} C_VEL
LIN {X 0,Y 262.556,Z 757.436,A -85,B 0,C 180,E1 -18236.792,E2 -18236.792} C_VEL
LIN {X 0,Y 261.771,Z 760.228,A -85,B 0,C 180,E1 -18239.33,E2 -18239.33} C_VEL
LIN {X 0,Y 261.052,Z 762.75,A -85,B 0,C 180,E1 -18242.764,E2 -18242.764} C_VEL
LIN {X 0,Y 260.737,Z 763.851,A -85,B 0,C 180,E1 -18246.153,E2 -18246.153} C_VEL
LIN {X 0,Y 260.724,Z 763.606,A -85,B 0,C 180,E1 -18249.488,E2 -18249.488} C_VEL
LIN {X 0,Y 260.888,Z 762.994,A -85,B 0,C 180,E1 -18251.141,E2 -18251.141} C_VEL
LIN {X 0,Y 261.205,Z 760.834,A -85,B 0,C 180,E1 -18254.393,E2 -18254.393} C_VEL
LIN {X 0,Y 261.909,Z 757.386,A -85,B 0,C 180,E1 -18257.605,E2 -18257.605} C_VEL
LIN {X 0,Y 262.95,Z 752.607,A -85,B 0,C 180,E1 -18260.773,E2 -18260.773} C_VEL
LIN {X 0,Y 264.464,Z 746.401,A -85,B 0,C 180,E1 -18263.899,E2 -18263.899} C_VEL
LIN {X 0,Y 266.591,Z 738.576,A -85,B 0,C 180,E1 -18266.979,E2 -18266.979} C_VEL
LIN {X 0,Y 268.844,Z 730.24,A -85,B 0,C 180,E1 -18269.626,E2 -18269.626} C_VEL
LIN {X 0,Y 271.622,Z 720.197,A -85,B 0,C 180,E1 -18272.225,E2 -18272.225} C_VEL
LIN {X 0,Y 274.722,Z 708.504,A -85,B 0,C 180,E1 -18274.676,E2 -18274.676} C_VEL
LIN {X 0,Y 277.692,Z 696.517,A -85,B 0,C 180,E1 -18276.723,E2 -18276.723} C_VEL
LIN {X 0,Y 280.574,Z 684.01,A -85,B 0,C 180,E1 -18278.463,E2 -18278.463} C_VEL
LIN {X 0,Y 283.308,Z 670.352,A -85,B 0,C 180,E1 -18280.001,E2 -18280.001} C_VEL
LIN {X 0,Y 285.66,Z 656.243,A -85,B 0,C 180,E1 -18281.262,E2 -18281.262} C_VEL
LIN {X 0,Y 287.551,Z 642.305,A -85,B 0,C 180,E1 -18282.224,E2 -18282.224} C_VEL
LIN {X 0,Y 289.139,Z 627.124,A -85,B 0,C 180,E1 -18282.987,E2 -18282.987} C_VEL
LIN {X 0,Y 290.146,Z 611.629,A -85,B 0,C 180,E1 -18283.501,E2 -18283.501} C_VEL
LIN {X 0,Y 294.417,Z 516.575,A -85,B 0,C 180,E1 -18285.803,E2 -18285.803} C_VEL
LIN {X 0,Y 294.181,Z 514.823,A -85,B 0,C 180,E1 -18285.889,E2 -18285.889} C_VEL
LIN {X 0,Y 285.868,Z 496.793,A -85,B 0,C 180,E1 -18287.649,E2 -18287.649} C_VEL
LIN {X 0,Y 279.781,Z 485.166,A -85,B 0,C 180,E1 -18288.975,E2 -18288.975} C_VEL
LIN {X 0,Y 270.516,Z 470.367,A -85,B 0,C 180,E1 -18291.042,E2 -18291.042} C_VEL
LIN {X 0,Y 267.399,Z 465.875,A -85,B 0,C 180,E1 -18291.761,E2 -18291.761} C_VEL
LIN {X 0,Y 265.453,Z 462.688,A -85,B 0,C 180,E1 -18292.236,E2 -18292.236} C_VEL
LIN {X 0,Y 263.736,Z 460.307,A -85,B 0,C 180,E1 -18292.649,E2 -18292.649} C_VEL
LIN {X 0,Y 263.195,Z 458.328,A -85,B 0,C 180,E1 -18292.833,E2 -18292.833} C_VEL
LIN {X 0,Y 263.213,Z 458.317,A -85,B 0,C 180,E1 -18295.291,E2 -18295.291} C_VEL
LIN {X 0,Y 263.17,Z 458.317,A -85,B 0,C 180,E1 -18298.731,E2 -18298.731} C_VEL
LIN {X 0,Y 263.137,Z 458.317,A -85,B 0,C 180,E1 -18302.288,E2 -18302.288} C_VEL
LIN {X 0,Y 263.167,Z 458.327,A -85,B 0,C 180,E1 -18305.982,E2 -18305.982} C_VEL
LIN {X 0,Y 263.134,Z 458.327,A -85,B 0,C 180,E1 -18309.868,E2 -18309.868} C_VEL
LIN {X 0,Y 263.127,Z 458.323,A -85,B 0,C 180,E1 -18313.984,E2 -18313.984} C_VEL
LIN {X 0,Y 263.157,Z 458.314,A -85,B 0,C 180,E1 -18318.399,E2 -18318.399} C_VEL
LIN {X 0,Y 263.191,Z 458.322,A -85,B 0,C 180,E1 -18322.108,E2 -18322.108} C_VEL
LIN {X 0,Y 263.187,Z 458.321,A -85,B 0,C 180,E1 -18325.89,E2 -18325.89} C_VEL
LIN {X 0,Y 263.143,Z 458.315,A -85,B 0,C 180,E1 -18329.505,E2 -18329.505} C_VEL
LIN {X 0,Y 263.181,Z 458.321,A -85,B 0,C 180,E1 -18332.537,E2 -18332.537} C_VEL
LIN {X 0,Y 262.535,Z 458.41,A -85,B 0,C 180,E1 -18333.813,E2 -18333.813} C_VEL
LIN {X 0,Y 259.715,Z 458.766,A -85,B 0,C 180,E1 -18335.894,E2 -18335.894} C_VEL
LIN {X 0,Y 257.301,Z 459.062,A -85,B 0,C 180,E1 -18337.586,E2 -18337.586} C_VEL
LIN {X 0,Y 256.249,Z 459.187,A -85,B 0,C 180,E1 -18338.897,E2 -18338.897} C_VEL
LIN {X 0,Y 256.155,Z 459.197,A -85,B 0,C 180,E1 -18339.342,E2 -18339.342} C_VEL
LIN {X 0,Y 256.302,Z 459.163,A -85,B 0,C 180,E1 -18344.085,E2 -18344.085} C_VEL
LIN {X 0,Y 256.312,Z 459.168,A -85,B 0,C 180,E1 -18348.934,E2 -18348.934} C_VEL
LIN {X 0,Y 256.542,Z 459.144,A -85,B 0,C 180,E1 -18352.127,E2 -18352.127} C_VEL
LIN {X 0,Y 256.715,Z 459.118,A -85,B 0,C 180,E1 -18358.431,E2 -18358.431} C_VEL
LIN {X 0,Y 256.716,Z 459.129,A -85,B 0,C 180,E1 -18361.568,E2 -18361.568} C_VEL
LIN {X 0,Y 256.541,Z 459.154,A -85,B 0,C 180,E1 -18367.873,E2 -18367.873} C_VEL
LIN {X 0,Y 256.311,Z 459.161,A -85,B 0,C 180,E1 -18371.066,E2 -18371.066} C_VEL
LIN {X 0,Y 256.301,Z 459.183,A -85,B 0,C 180,E1 -18375.914,E2 -18375.914} C_VEL
LIN {X 0,Y 256.219,Z 459.192,A -85,B 0,C 180,E1 -18380.89,E2 -18380.89} C_VEL
LIN {X 0,Y 256.19,Z 459.197,A -85,B 0,C 180,E1 -18385.138,E2 -18385.138} C_VEL
LIN {X 0,Y 256.112,Z 459.208,A -85,B 0,C 180,E1 -18389.599,E2 -18389.599} C_VEL
LIN {X 0,Y 256.086,Z 459.207,A -85,B 0,C 180,E1 -18393.29,E2 -18393.29} C_VEL
LIN {X 0,Y 256.129,Z 459.206,A -85,B 0,C 180,E1 -18397.274,E2 -18397.274} C_VEL
LIN {X 0,Y 256.107,Z 459.305,A -85,B 0,C 180,E1 -18401.3,E2 -18401.3} C_VEL
LIN {X 0,Y 258.314,Z 466.332,A -85,B 0,C 180,E1 -18404.112,E2 -18404.112} C_VEL
LIN {X 0,Y 267.048,Z 481.459,A -85,B 0,C 180,E1 -18406.327,E2 -18406.327} C_VEL
LIN {X 0,Y 275.757,Z 498.231,A -85,B 0,C 180,E1 -18408.405,E2 -18408.405} C_VEL
LIN {X 0,Y 283.699,Z 515.576,A -85,B 0,C 180,E1 -18410.224,E2 -18410.224} C_VEL
LIN {X 0,Y 288.022,Z 526.086,A -85,B 0,C 180,E1 -18411.189,E2 -18411.189} C_VEL
LIN {X 0,Y 288.285,Z 528.944,A -85,B 0,C 180,E1 -18411.316,E2 -18411.316} C_VEL
LIN {X 0,Y 283.421,Z 633.086,A -85,B 0,C 180,E1 -18413.919,E2 -18413.919} C_VEL
LIN {X 0,Y 281.92,Z 649.16,A -85,B 0,C 180,E1 -18414.577,E2 -18414.577} C_VEL
LIN {X 0,Y 279.788,Z 664.401,A -85,B 0,C 180,E1 -18415.476,E2 -18415.476} C_VEL
LIN {X 0,Y 277.314,Z 679.086,A -85,B 0,C 180,E1 -18416.657,E2 -18416.657} C_VEL
LIN {X 0,Y 274.764,Z 691.701,A -85,B 0,C 180,E1 -18417.943,E2 -18417.943} C_VEL
LIN {X 0,Y 271.576,Z 705.473,A -85,B 0,C 180,E1 -18419.693,E2 -18419.693} C_VEL
LIN {X 0,Y 268.423,Z 717.951,A -85,B 0,C 180,E1 -18421.669,E2 -18421.669} C_VEL
LIN {X 0,Y 265.508,Z 728.588,A -85,B 0,C 180,E1 -18423.722,E2 -18423.722} C_VEL
LIN {X 0,Y 262.95,Z 738.178,A -85,B 0,C 180,E1 -18425.963,E2 -18425.963} C_VEL
LIN {X 0,Y 260.189,Z 747.629,A -85,B 0,C 180,E1 -18428.613,E2 -18428.613} C_VEL
LIN {X 0,Y 258.104,Z 755.546,A -85,B 0,C 180,E1 -18431.34,E2 -18431.34} C_VEL
LIN {X 0,Y 256.401,Z 762.097,A -85,B 0,C 180,E1 -18434.091,E2 -18434.091} C_VEL
LIN {X 0,Y 255.104,Z 768.105,A -85,B 0,C 180,E1 -18437.267,E2 -18437.267} C_VEL
LIN {X 0,Y 254.339,Z 772.711,A -85,B 0,C 180,E1 -18440.456,E2 -18440.456} C_VEL
LIN {X 0,Y 254.037,Z 775.998,A -85,B 0,C 180,E1 -18443.646,E2 -18443.646} C_VEL
LIN {X 0,Y 253.937,Z 778.024,A -85,B 0,C 180,E1 -18446.826,E2 -18446.826} C_VEL
LIN {X 0,Y 254.053,Z 778.875,A -85,B 0,C 180,E1 -18449.999,E2 -18449.999} C_VEL
LIN {X 0,Y 253.938,Z 778.563,A -85,B 0,C 180,E1 -18453.172,E2 -18453.172} C_VEL
LIN {X 0,Y 253.993,Z 777.103,A -85,B 0,C 180,E1 -18456.354,E2 -18456.354} C_VEL
LIN {X 0,Y 254.341,Z 774.443,A -85,B 0,C 180,E1 -18459.542,E2 -18459.542} C_VEL
LIN {X 0,Y 255.153,Z 770.54,A -85,B 0,C 180,E1 -18462.729,E2 -18462.729} C_VEL
LIN {X 0,Y 256.528,Z 765.344,A -85,B 0,C 180,E1 -18465.899,E2 -18465.899} C_VEL
LIN {X 0,Y 258.53,Z 758.724,A -85,B 0,C 180,E1 -18469.038,E2 -18469.038} C_VEL
LIN {X 0,Y 261.227,Z 750.501,A -85,B 0,C 180,E1 -18472.125,E2 -18472.125} C_VEL
LIN {X 0,Y 264.338,Z 741.76,A -85,B 0,C 180,E1 -18474.754,E2 -18474.754} C_VEL
LIN {X 0,Y 267.13,Z 732.914,A -85,B 0,C 180,E1 -18476.989,E2 -18476.989} C_VEL
LIN {X 0,Y 270.548,Z 722.516,A -85,B 0,C 180,E1 -18479.147,E2 -18479.147} C_VEL
LIN {X 0,Y 274.291,Z 710.119,A -85,B 0,C 180,E1 -18481.254,E2 -18481.254} C_VEL
LIN {X 0,Y 277.747,Z 697.736,A -85,B 0,C 180,E1 -18482.957,E2 -18482.957} C_VEL
LIN {X 0,Y 281.136,Z 683.554,A -85,B 0,C 180,E1 -18484.527,E2 -18484.527} C_VEL
LIN {X 0,Y 284.068,Z 669.226,A -85,B 0,C 180,E1 -18485.766,E2 -18485.766} C_VEL
LIN {X 0,Y 286.591,Z 654.702,A -85,B 0,C 180,E1 -18486.707,E2 -18486.707} C_VEL
LIN {X 0,Y 288.537,Z 639.887,A -85,B 0,C 180,E1 -18487.401,E2 -18487.401} C_VEL
LIN {X 0,Y 289.703,Z 624.906,A -85,B 0,C 180,E1 -18487.883,E2 -18487.883} C_VEL
LIN {X 0,Y 294.192,Z 539.52,A -85,B 0,C 180,E1 -18489.984,E2 -18489.984} C_VEL
LIN {X 0,Y 294.636,Z 529.612,A -85,B 0,C 180,E1 -18490.244,E2 -18490.244} C_VEL
LIN {X 0,Y 288.17,Z 514.529,A -85,B 0,C 180,E1 -18492.039,E2 -18492.039} C_VEL
LIN {X 0,Y 280.977,Z 500.233,A -85,B 0,C 180,E1 -18494.135,E2 -18494.135} C_VEL
LIN {X 0,Y 274.944,Z 489.728,A -85,B 0,C 180,E1 -18496.02,E2 -18496.02} C_VEL
LIN {X 0,Y 269,Z 480.348,A -85,B 0,C 180,E1 -18498.01,E2 -18498.01} C_VEL
LIN {X 0,Y 265.53,Z 475.172,A -85,B 0,C 180,E1 -18499.263,E2 -18499.263} C_VEL
LIN {X 0,Y 261.685,Z 469.595,A -85,B 0,C 180,E1 -18500.751,E2 -18500.751} C_VEL
LIN {X 0,Y 257.742,Z 463.981,A -85,B 0,C 180,E1 -18502.422,E2 -18502.422} C_VEL
LIN {X 0,Y 256.114,Z 459.206,A -85,B 0,C 180,E1 -18505.407,E2 -18505.407} C_VEL
LIN {X 0,Y 256.086,Z 459.212,A -85,B 0,C 180,E1 -18508.572,E2 -18508.572} C_VEL
LIN {X 0,Y 256.135,Z 459.2,A -85,B 0,C 180,E1 -18512.196,E2 -18512.196} C_VEL
LIN {X 0,Y 256.161,Z 459.194,A -85,B 0,C 180,E1 -18515.699,E2 -18515.699} C_VEL
LIN {X 0,Y 256.161,Z 459.193,A -85,B 0,C 180,E1 -18519.105,E2 -18519.105} C_VEL
LIN {X 0,Y 256.294,Z 459.178,A -85,B 0,C 180,E1 -18524.085,E2 -18524.085} C_VEL
LIN {X 0,Y 256.304,Z 459.183,A -85,B 0,C 180,E1 -18528.934,E2 -18528.934} C_VEL
LIN {X 0,Y 256.534,Z 459.156,A -85,B 0,C 180,E1 -18532.127,E2 -18532.127} C_VEL
LIN {X 0,Y 256.709,Z 459.125,A -85,B 0,C 180,E1 -18538.432,E2 -18538.432} C_VEL
LIN {X 0,Y 256.709,Z 459.123,A -85,B 0,C 180,E1 -18541.569,E2 -18541.569} C_VEL
LIN {X 0,Y 256.534,Z 459.147,A -85,B 0,C 180,E1 -18547.874,E2 -18547.874} C_VEL
LIN {X 0,Y 256.304,Z 459.176,A -85,B 0,C 180,E1 -18551.067,E2 -18551.067} C_VEL
LIN {X 0,Y 256.317,Z 459.322,A -85,B 0,C 180,E1 -18555.303,E2 -18555.303} C_VEL
LIN {X 0,Y 257.176,Z 461.828,A -85,B 0,C 180,E1 -18555.758,E2 -18555.758} C_VEL
LIN {X 0,Y 259.269,Z 464.159,A -85,B 0,C 180,E1 -18556.618,E2 -18556.618} C_VEL
LIN {X 0,Y 260.384,Z 465.071,A -85,B 0,C 180,E1 -18557.044,E2 -18557.044} C_VEL
LIN {X 0,Y 262.314,Z 468.258,A -85,B 0,C 180,E1 -18557.845,E2 -18557.845} C_VEL
LIN {X 0,Y 264.382,Z 470.263,A -85,B 0,C 180,E1 -18558.602,E2 -18558.602} C_VEL
LIN {X 0,Y 266.834,Z 473.834,A -85,B 0,C 180,E1 -18559.522,E2 -18559.522} C_VEL
LIN {X 0,Y 268.25,Z 475.679,A -85,B 0,C 180,E1 -18560.024,E2 -18560.024} C_VEL
LIN {X 0,Y 272.172,Z 480.969,A -85,B 0,C 180,E1 -18561.342,E2 -18561.342} C_VEL
LIN {X 0,Y 277.23,Z 488.049,A -85,B 0,C 180,E1 -18562.941,E2 -18562.941} C_VEL
LIN {X 0,Y 282.132,Z 495.931,A -85,B 0,C 180,E1 -18564.416,E2 -18564.416} C_VEL
LIN {X 0,Y 288.328,Z 507.339,A -85,B 0,C 180,E1 -18566.189,E2 -18566.189} C_VEL
LIN {X 0,Y 294.263,Z 519.893,A -85,B 0,C 180,E1 -18567.805,E2 -18567.805} C_VEL
LIN {X 0,Y 295.026,Z 521.553,A -85,B 0,C 180,E1 -18568.007,E2 -18568.007} C_VEL
LIN {X 0,Y 289.743,Z 620.137,A -85,B 0,C 180,E1 -18570.472,E2 -18570.472} C_VEL
LIN {X 0,Y 288.065,Z 635.988,A -85,B 0,C 180,E1 -18571.11,E2 -18571.11} C_VEL
LIN {X 0,Y 285.949,Z 651.063,A -85,B 0,C 180,E1 -18572.015,E2 -18572.015} C_VEL
LIN {X 0,Y 283.29,Z 665.846,A -85,B 0,C 180,E1 -18573.209,E2 -18573.209} C_VEL
LIN {X 0,Y 280.17,Z 679.909,A -85,B 0,C 180,E1 -18574.661,E2 -18574.661} C_VEL
LIN {X 0,Y 276.854,Z 692.644,A -85,B 0,C 180,E1 -18576.297,E2 -18576.297} C_VEL
LIN {X 0,Y 273.487,Z 704.481,A -85,B 0,C 180,E1 -18578.182,E2 -18578.182} C_VEL
LIN {X 0,Y 269.91,Z 715.853,A -85,B 0,C 180,E1 -18580.396,E2 -18580.396} C_VEL
LIN {X 0,Y 266.568,Z 725.862,A -85,B 0,C 180,E1 -18582.779,E2 -18582.779} C_VEL
LIN {X 0,Y 263.254,Z 735.223,A -85,B 0,C 180,E1 -18585.512,E2 -18585.512} C_VEL
LIN {X 0,Y 260.341,Z 743.545,A -85,B 0,C 180,E1 -18588.557,E2 -18588.557} C_VEL
LIN {X 0,Y 258.265,Z 749.44,A -85,B 0,C 180,E1 -18591.255,E2 -18591.255} C_VEL
LIN {X 0,Y 256.655,Z 754.163,A -85,B 0,C 180,E1 -18593.934,E2 -18593.934} C_VEL
LIN {X 0,Y 255.513,Z 757.931,A -85,B 0,C 180,E1 -18596.627,E2 -18596.627} C_VEL
LIN {X 0,Y 254.863,Z 760.193,A -85,B 0,C 180,E1 -18598.743,E2 -18598.743} C_VEL
LIN {X 0,Y 254.036,Z 762.835,A -85,B 0,C 180,E1 -18602.288,E2 -18602.288} C_VEL
LIN {X 0,Y 253.664,Z 764.005,A -85,B 0,C 180,E1 -18605.445,E2 -18605.445} C_VEL
LIN {X 0,Y 253.597,Z 763.974,A -85,B 0,C 180,E1 -18608.884,E2 -18608.884} C_VEL
LIN {X 0,Y 253.749,Z 763.46,A -85,B 0,C 180,E1 -18610.589,E2 -18610.589} C_VEL
LIN {X 0,Y 254.042,Z 761.488,A -85,B 0,C 180,E1 -18613.941,E2 -18613.941} C_VEL
LIN {X 0,Y 254.732,Z 758.234,A -85,B 0,C 180,E1 -18617.25,E2 -18617.25} C_VEL
LIN {X 0,Y 255.735,Z 753.676,A -85,B 0,C 180,E1 -18620.51,E2 -18620.51} C_VEL
LIN {X 0,Y 257.237,Z 747.716,A -85,B 0,C 180,E1 -18623.727,E2 -18623.727} C_VEL
LIN {X 0,Y 259.374,Z 740.178,A -85,B 0,C 180,E1 -18626.894,E2 -18626.894} C_VEL
LIN {X 0,Y 261.649,Z 732.114,A -85,B 0,C 180,E1 -18629.616,E2 -18629.616} C_VEL
LIN {X 0,Y 264.448,Z 722.414,A -85,B 0,C 180,E1 -18632.285,E2 -18632.285} C_VEL
LIN {X 0,Y 267.22,Z 712.51,A -85,B 0,C 180,E1 -18634.526,E2 -18634.526} C_VEL
LIN {X 0,Y 270.32,Z 700.738,A -85,B 0,C 180,E1 -18636.719,E2 -18636.719} C_VEL
LIN {X 0,Y 273.526,Z 687.71,A -85,B 0,C 180,E1 -18638.683,E2 -18638.683} C_VEL
LIN {X 0,Y 276.287,Z 674.832,A -85,B 0,C 180,E1 -18640.258,E2 -18640.258} C_VEL
LIN {X 0,Y 278.824,Z 660.793,A -85,B 0,C 180,E1 -18641.634,E2 -18641.634} C_VEL
LIN {X 0,Y 280.99,Z 646.458,A -85,B 0,C 180,E1 -18642.72,E2 -18642.72} C_VEL
LIN {X 0,Y 282.747,Z 631.034,A -85,B 0,C 180,E1 -18643.587,E2 -18643.587} C_VEL
LIN {X 0,Y 283.988,Z 615.717,A -85,B 0,C 180,E1 -18644.16,E2 -18644.16} C_VEL
LIN {X 0,Y 288.578,Z 517.899,A -85,B 0,C 180,E1 -18646.584,E2 -18646.584} C_VEL
LIN {X 0,Y 284.84,Z 509.069,A -85,B 0,C 180,E1 -18647.41,E2 -18647.41} C_VEL
LIN {X 0,Y 276.392,Z 491.824,A -85,B 0,C 180,E1 -18649.303,E2 -18649.303} C_VEL
LIN {X 0,Y 266.452,Z 475.629,A -85,B 0,C 180,E1 -18651.581,E2 -18651.581} C_VEL
LIN {X 0,Y 260.819,Z 467.244,A -85,B 0,C 180,E1 -18652.953,E2 -18652.953} C_VEL
LIN {X 0,Y 258.349,Z 463.487,A -85,B 0,C 180,E1 -18653.582,E2 -18653.582} C_VEL
LIN {X 0,Y 256.639,Z 461.052,A -85,B 0,C 180,E1 -18654.02,E2 -18654.02} C_VEL
LIN {X 0,Y 256.149,Z 459.193,A -85,B 0,C 180,E1 -18654.203,E2 -18654.203} C_VEL
LIN {X 0,Y 256.131,Z 459.193,A -85,B 0,C 180,E1 -18658.591,E2 -18658.591} C_VEL
LIN {X 0,Y 256.086,Z 459.199,A -85,B 0,C 180,E1 -18661.705,E2 -18661.705} C_VEL
LIN {X 0,Y 256.112,Z 459.21,A -85,B 0,C 180,E1 -18665.189,E2 -18665.189} C_VEL
LIN {X 0,Y 256.097,Z 459.195,A -85,B 0,C 180,E1 -18669.138,E2 -18669.138} C_VEL
LIN {X 0,Y 256.067,Z 459.2,A -85,B 0,C 180,E1 -18673.326,E2 -18673.326} C_VEL
LIN {X 0,Y 256.093,Z 459.196,A -85,B 0,C 180,E1 -18677.814,E2 -18677.814} C_VEL
LIN {X 0,Y 256.103,Z 459.208,A -85,B 0,C 180,E1 -18680.863,E2 -18680.863} C_VEL
LIN {X 0,Y 256.124,Z 459.191,A -85,B 0,C 180,E1 -18684.813,E2 -18684.813} C_VEL
LIN {X 0,Y 256.095,Z 459.202,A -85,B 0,C 180,E1 -18688.572,E2 -18688.572} C_VEL
LIN {X 0,Y 256.121,Z 459.2,A -85,B 0,C 180,E1 -18692.521,E2 -18692.521} C_VEL
LIN {X 0,Y 256.145,Z 459.185,A -85,B 0,C 180,E1 -18695.696,E2 -18695.696} C_VEL
LIN {X 0,Y 256.155,Z 459.197,A -85,B 0,C 180,E1 -18699.342,E2 -18699.342} C_VEL
LIN {X 0,Y 255.468,Z 459.286,A -85,B 0,C 180,E1 -18700.656,E2 -18700.656} C_VEL
LIN {X 0,Y 252.632,Z 459.625,A -85,B 0,C 180,E1 -18702.799,E2 -18702.799} C_VEL
LIN {X 0,Y 250.256,Z 459.922,A -85,B 0,C 180,E1 -18704.543,E2 -18704.543} C_VEL
LIN {X 0,Y 249.263,Z 460.056,A -85,B 0,C 180,E1 -18705.895,E2 -18705.895} C_VEL
LIN {X 0,Y 249.194,Z 460.062,A -85,B 0,C 180,E1 -18706.352,E2 -18706.352} C_VEL
LIN {X 0,Y 249.427,Z 460.016,A -85,B 0,C 180,E1 -18710.465,E2 -18710.465} C_VEL
LIN {X 0,Y 249.463,Z 460.036,A -85,B 0,C 180,E1 -18713.529,E2 -18713.529} C_VEL
LIN {X 0,Y 249.677,Z 459.994,A -85,B 0,C 180,E1 -18718.387,E2 -18718.387} C_VEL
LIN {X 0,Y 249.677,Z 460.005,A -85,B 0,C 180,E1 -18721.613,E2 -18721.613} C_VEL
LIN {X 0,Y 249.463,Z 460.02,A -85,B 0,C 180,E1 -18726.47,E2 -18726.47} C_VEL
LIN {X 0,Y 249.39,Z 460.037,A -85,B 0,C 180,E1 -18729.734,E2 -18729.734} C_VEL
LIN {X 0,Y 249.207,Z 460.066,A -85,B 0,C 180,E1 -18734.703,E2 -18734.703} C_VEL
LIN {X 0,Y 249.141,Z 460.054,A -85,B 0,C 180,E1 -18738.077,E2 -18738.077} C_VEL
LIN {X 0,Y 249.105,Z 460.082,A -85,B 0,C 180,E1 -18741.516,E2 -18741.516} C_VEL
LIN {X 0,Y 249.132,Z 460.074,A -85,B 0,C 180,E1 -18745.482,E2 -18745.482} C_VEL
LIN {X 0,Y 249.082,Z 460.08,A -85,B 0,C 180,E1 -18748.992,E2 -18748.992} C_VEL
LIN {X 0,Y 249.037,Z 460.089,A -85,B 0,C 180,E1 -18752.424,E2 -18752.424} C_VEL
LIN {X 0,Y 249.07,Z 460.082,A -85,B 0,C 180,E1 -18756.338,E2 -18756.338} C_VEL
LIN {X 0,Y 249.021,Z 460.091,A -85,B 0,C 180,E1 -18760.067,E2 -18760.067} C_VEL
LIN {X 0,Y 250.98,Z 466.153,A -85,B 0,C 180,E1 -18762.596,E2 -18762.596} C_VEL
LIN {X 0,Y 253.711,Z 470.684,A -85,B 0,C 180,E1 -18763.346,E2 -18763.346} C_VEL
LIN {X 0,Y 262.462,Z 485.869,A -85,B 0,C 180,E1 -18765.646,E2 -18765.646} C_VEL
LIN {X 0,Y 271.823,Z 504.161,A -85,B 0,C 180,E1 -18767.957,E2 -18767.957} C_VEL
LIN {X 0,Y 280.431,Z 523.601,A -85,B 0,C 180,E1 -18769.99,E2 -18769.99} C_VEL
LIN {X 0,Y 282.48,Z 528.776,A -85,B 0,C 180,E1 -18770.468,E2 -18770.468} C_VEL
LIN {X 0,Y 277.743,Z 628.837,A -85,B 0,C 180,E1 -18773.004,E2 -18773.004} C_VEL
LIN {X 0,Y 276.407,Z 644.715,A -85,B 0,C 180,E1 -18773.591,E2 -18773.591} C_VEL
LIN {X 0,Y 274.507,Z 659.248,A -85,B 0,C 180,E1 -18774.376,E2 -18774.376} C_VEL
LIN {X 0,Y 272.239,Z 673.117,A -85,B 0,C 180,E1 -18775.393,E2 -18775.393} C_VEL
LIN {X 0,Y 269.758,Z 685.904,A -85,B 0,C 180,E1 -18776.589,E2 -18776.589} C_VEL
LIN {X 0,Y 266.699,Z 699.511,A -85,B 0,C 180,E1 -18778.194,E2 -18778.194} C_VEL
LIN {X 0,Y 263.616,Z 711.895,A -85,B 0,C 180,E1 -18780.008,E2 -18780.008} C_VEL
LIN {X 0,Y 260.109,Z 724.22,A -85,B 0,C 180,E1 -18782.219,E2 -18782.219} C_VEL
LIN {X 0,Y 257.111,Z 734.847,A -85,B 0,C 180,E1 -18784.574,E2 -18784.574} C_VEL
LIN {X 0,Y 254.357,Z 744.681,A -85,B 0,C 180,E1 -18787.242,E2 -18787.242} C_VEL
LIN {X 0,Y 251.849,Z 753.052,A -85,B 0,C 180,E1 -18790.01,E2 -18790.01} C_VEL
LIN {X 0,Y 249.758,Z 760.563,A -85,B 0,C 180,E1 -18793.083,E2 -18793.083} C_VEL
LIN {X 0,Y 248.415,Z 766.392,A -85,B 0,C 180,E1 -18796.085,E2 -18796.085} C_VEL
LIN {X 0,Y 247.429,Z 771.351,A -85,B 0,C 180,E1 -18799.36,E2 -18799.36} C_VEL
LIN {X 0,Y 247.078,Z 774.236,A -85,B 0,C 180,E1 -18801.823,E2 -18801.823} C_VEL
LIN {X 0,Y 246.841,Z 776.977,A -85,B 0,C 180,E1 -18805.209,E2 -18805.209} C_VEL
LIN {X 0,Y 246.92,Z 778.366,A -85,B 0,C 180,E1 -18808.368,E2 -18808.368} C_VEL
LIN {X 0,Y 246.982,Z 778.661,A -85,B 0,C 180,E1 -18809.999,E2 -18809.999} C_VEL
LIN {X 0,Y 246.84,Z 778.375,A -85,B 0,C 180,E1 -18813.263,E2 -18813.263} C_VEL
LIN {X 0,Y 246.9,Z 776.942,A -85,B 0,C 180,E1 -18816.537,E2 -18816.537} C_VEL
LIN {X 0,Y 247.297,Z 774.3,A -85,B 0,C 180,E1 -18819.817,E2 -18819.817} C_VEL
LIN {X 0,Y 248.189,Z 770.434,A -85,B 0,C 180,E1 -18823.092,E2 -18823.092} C_VEL
LIN {X 0,Y 249.615,Z 765.273,A -85,B 0,C 180,E1 -18826.352,E2 -18826.352} C_VEL
LIN {X 0,Y 251.76,Z 758.691,A -85,B 0,C 180,E1 -18829.57,E2 -18829.57} C_VEL
LIN {X 0,Y 254.616,Z 750.507,A -85,B 0,C 180,E1 -18832.732,E2 -18832.732} C_VEL
LIN {X 0,Y 257.857,Z 741.82,A -85,B 0,C 180,E1 -18835.42,E2 -18835.42} C_VEL
LIN {X 0,Y 260.795,Z 733.048,A -85,B 0,C 180,E1 -18837.7,E2 -18837.7} C_VEL
LIN {X 0,Y 264.359,Z 722.74,A -85,B 0,C 180,E1 -18839.897,E2 -18839.897} C_VEL
LIN {X 0,Y 268.259,Z 710.43,A -85,B 0,C 180,E1 -18842.039,E2 -18842.039} C_VEL
LIN {X 0,Y 271.835,Z 698.142,A -85,B 0,C 180,E1 -18843.768,E2 -18843.768} C_VEL
LIN {X 0,Y 275.31,Z 684.327,A -85,B 0,C 180,E1 -18845.337,E2 -18845.337} C_VEL
LIN {X 0,Y 278.373,Z 669.997,A -85,B 0,C 180,E1 -18846.615,E2 -18846.615} C_VEL
LIN {X 0,Y 280.966,Z 655.749,A -85,B 0,C 180,E1 -18847.567,E2 -18847.567} C_VEL
LIN {X 0,Y 283.089,Z 640.497,A -85,B 0,C 180,E1 -18848.306,E2 -18848.306} C_VEL
LIN {X 0,Y 284.403,Z 624.553,A -85,B 0,C 180,E1 -18848.831,E2 -18848.831} C_VEL
LIN {X 0,Y 289.008,Z 541.067,A -85,B 0,C 180,E1 -18850.913,E2 -18850.913} C_VEL
LIN {X 0,Y 289.4,Z 531.901,A -85,B 0,C 180,E1 -18851.165,E2 -18851.165} C_VEL
LIN {X 0,Y 283.395,Z 517.833,A -85,B 0,C 180,E1 -18852.915,E2 -18852.915} C_VEL
LIN {X 0,Y 277.103,Z 505.095,A -85,B 0,C 180,E1 -18854.843,E2 -18854.843} C_VEL
LIN {X 0,Y 270.533,Z 493.422,A -85,B 0,C 180,E1 -18857.006,E2 -18857.006} C_VEL
LIN {X 0,Y 265.065,Z 484.779,A -85,B 0,C 180,E1 -18858.941,E2 -18858.941} C_VEL
LIN {X 0,Y 262.439,Z 480.779,A -85,B 0,C 180,E1 -18859.944,E2 -18859.944} C_VEL
LIN {X 0,Y 258.901,Z 475.546,A -85,B 0,C 180,E1 -18861.366,E2 -18861.366} C_VEL
LIN {X 0,Y 254.226,Z 469.042,A -85,B 0,C 180,E1 -18863.391,E2 -18863.391} C_VEL
LIN {X 0,Y 250.632,Z 464.252,A -85,B 0,C 180,E1 -18865.123,E2 -18865.123} C_VEL
LIN {X 0,Y 250.299,Z 463.509,A -85,B 0,C 180,E1 -18865.363,E2 -18865.363} C_VEL
LIN {X 0,Y 249.033,Z 460.086,A -85,B 0,C 180,E1 -18867.845,E2 -18867.845} C_VEL
LIN {X 0,Y 249.091,Z 460.084,A -85,B 0,C 180,E1 -18871.338,E2 -18871.338} C_VEL
LIN {X 0,Y 249.145,Z 460.074,A -85,B 0,C 180,E1 -18874.968,E2 -18874.968} C_VEL
LIN {X 0,Y 249.104,Z 460.072,A -85,B 0,C 180,E1 -18880.211,E2 -18880.211} C_VEL
LIN {X 0,Y 249.236,Z 460.054,A -85,B 0,C 180,E1 -18883.622,E2 -18883.622} C_VEL
LIN {X 0,Y 249.247,Z 460.064,A -85,B 0,C 180,E1 -18888.617,E2 -18888.617} C_VEL
LIN {X 0,Y 249.475,Z 460.033,A -85,B 0,C 180,E1 -18891.903,E2 -18891.903} C_VEL
LIN {X 0,Y 249.432,Z 460.034,A -85,B 0,C 180,E1 -18896.77,E2 -18896.77} C_VEL
LIN {X 0,Y 249.722,Z 460.002,A -85,B 0,C 180,E1 -18900,E2 -18900} C_VEL
LIN {X 0,Y 249.432,Z 460.041,A -85,B 0,C 180,E1 -18903.231,E2 -18903.231} C_VEL
LIN {X 0,Y 249.476,Z 460.026,A -85,B 0,C 180,E1 -18908.098,E2 -18908.098} C_VEL
LIN {X 0,Y 249.247,Z 460.064,A -85,B 0,C 180,E1 -18912.468,E2 -18912.468} C_VEL
LIN {X 0,Y 250.06,Z 462.637,A -85,B 0,C 180,E1 -18912.994,E2 -18912.994} C_VEL
LIN {X 0,Y 251.959,Z 464.848,A -85,B 0,C 180,E1 -18913.921,E2 -18913.921} C_VEL
LIN {X 0,Y 253.658,Z 465.949,A -85,B 0,C 180,E1 -18914.666,E2 -18914.666} C_VEL
LIN {X 0,Y 255.47,Z 469.094,A -85,B 0,C 180,E1 -18915.539,E2 -18915.539} C_VEL
LIN {X 0,Y 257.755,Z 471.456,A -85,B 0,C 180,E1 -18916.486,E2 -18916.486} C_VEL
LIN {X 0,Y 260.32,Z 475.051,A -85,B 0,C 180,E1 -18917.542,E2 -18917.542} C_VEL
LIN {X 0,Y 261.745,Z 476.641,A -85,B 0,C 180,E1 -18918.087,E2 -18918.087} C_VEL
LIN {X 0,Y 265.758,Z 482.284,A -85,B 0,C 180,E1 -18919.605,E2 -18919.605} C_VEL
LIN {X 0,Y 268.988,Z 486.631,A -85,B 0,C 180,E1 -18920.732,E2 -18920.732} C_VEL
LIN {X 0,Y 274.012,Z 493.836,A -85,B 0,C 180,E1 -18922.379,E2 -18922.379} C_VEL
LIN {X 0,Y 278.56,Z 501.343,A -85,B 0,C 180,E1 -18923.809,E2 -18923.809} C_VEL
LIN {X 0,Y 284.424,Z 512.443,A -85,B 0,C 180,E1 -18925.56,E2 -18925.56} C_VEL
LIN {X 0,Y 289.831,Z 524.118,A -85,B 0,C 180,E1 -18927.099,E2 -18927.099} C_VEL
LIN {X 0,Y 284.448,Z 620.233,A -85,B 0,C 180,E1 -18929.533,E2 -18929.533} C_VEL
LIN {X 0,Y 282.723,Z 635.94,A -85,B 0,C 180,E1 -18930.165,E2 -18930.165} C_VEL
LIN {X 0,Y 280.541,Z 651.051,A -85,B 0,C 180,E1 -18931.082,E2 -18931.082} C_VEL
LIN {X 0,Y 277.946,Z 664.989,A -85,B 0,C 180,E1 -18932.204,E2 -18932.204} C_VEL
LIN {X 0,Y 275.035,Z 677.937,A -85,B 0,C 180,E1 -18933.526,E2 -18933.526} C_VEL
LIN {X 0,Y 271.688,Z 690.547,A -85,B 0,C 180,E1 -18935.11,E2 -18935.11} C_VEL
LIN {X 0,Y 268.038,Z 703.162,A -85,B 0,C 180,E1 -18937.09,E2 -18937.09} C_VEL
LIN {X 0,Y 264.331,Z 714.434,A -85,B 0,C 180,E1 -18939.254,E2 -18939.254} C_VEL
LIN {X 0,Y 260.903,Z 724.311,A -85,B 0,C 180,E1 -18941.577,E2 -18941.577} C_VEL
LIN {X 0,Y 257.488,Z 733.582,A -85,B 0,C 180,E1 -18944.237,E2 -18944.237} C_VEL
LIN {X 0,Y 254.635,Z 741.192,A -85,B 0,C 180,E1 -18946.915,E2 -18946.915} C_VEL
LIN {X 0,Y 251.922,Z 748.434,A -85,B 0,C 180,E1 -18950.087,E2 -18950.087} C_VEL
LIN {X 0,Y 250.153,Z 753.45,A -85,B 0,C 180,E1 -18952.842,E2 -18952.842} C_VEL
LIN {X 0,Y 248.461,Z 758.482,A -85,B 0,C 180,E1 -18956.526,E2 -18956.526} C_VEL
LIN {X 0,Y 247.595,Z 761.17,A -85,B 0,C 180,E1 -18959.276,E2 -18959.276} C_VEL
LIN {X 0,Y 246.833,Z 763.451,A -85,B 0,C 180,E1 -18962.9,E2 -18962.9} C_VEL
LIN {X 0,Y 246.532,Z 764.319,A -85,B 0,C 180,E1 -18966.479,E2 -18966.479} C_VEL
LIN {X 0,Y 246.602,Z 763.807,A -85,B 0,C 180,E1 -18970.134,E2 -18970.134} C_VEL
LIN {X 0,Y 246.866,Z 762.096,A -85,B 0,C 180,E1 -18973.461,E2 -18973.461} C_VEL
LIN {X 0,Y 247.536,Z 759.067,A -85,B 0,C 180,E1 -18976.873,E2 -18976.873} C_VEL
LIN {X 0,Y 248.503,Z 754.743,A -85,B 0,C 180,E1 -18980.231,E2 -18980.231} C_VEL
LIN {X 0,Y 250.024,Z 749.022,A -85,B 0,C 180,E1 -18983.545,E2 -18983.545} C_VEL
LIN {X 0,Y 252.135,Z 741.754,A -85,B 0,C 180,E1 -18986.805,E2 -18986.805} C_VEL
LIN {X 0,Y 254.419,Z 733.982,A -85,B 0,C 180,E1 -18989.605,E2 -18989.605} C_VEL
LIN {X 0,Y 257.283,Z 724.599,A -85,B 0,C 180,E1 -18992.349,E2 -18992.349} C_VEL
LIN {X 0,Y 260.04,Z 715.091,A -85,B 0,C 180,E1 -18994.651,E2 -18994.651} C_VEL
LIN {X 0,Y 263.17,Z 703.776,A -85,B 0,C 180,E1 -18996.903,E2 -18996.903} C_VEL
LIN {X 0,Y 266.43,Z 691.315,A -85,B 0,C 180,E1 -18998.916,E2 -18998.916} C_VEL
LIN {X 0,Y 269.587,Z 677.588,A -85,B 0,C 180,E1 -19000.705,E2 -19000.705} C_VEL
LIN {X 0,Y 272.245,Z 663.973,A -85,B 0,C 180,E1 -19002.127,E2 -19002.127} C_VEL
LIN {X 0,Y 274.586,Z 649.357,A -85,B 0,C 180,E1 -19003.319,E2 -19003.319} C_VEL
LIN {X 0,Y 276.562,Z 633.611,A -85,B 0,C 180,E1 -19004.263,E2 -19004.263} C_VEL
LIN {X 0,Y 277.962,Z 618.395,A -85,B 0,C 180,E1 -19004.879,E2 -19004.879} C_VEL
